# B&R Automation Studio project ABC_Pltzr (part 2)

#### bgTelnetSrvr-astcpV2.c
```c
#include <bur/plctypes.h>

#ifdef _DEFAULT_INCLUDES
	#include <AsDefault.h>
#endif
/*
File: bgTelnetSrvr-astcpV2.c
=====

Modified on June 2015:
-modifications and adjustements to the latest version of bglib and B&R libraries

Modified on Jyly 2007:
THIS IS AN UPDATED VERSION OF THE TELNET SERVER WITH A SUPPORT FOR NEW B&R TCP LIBRARY!
OLD B&R TCP LIBRARY: ETHERNET.LIB
NEW B&R TCP LIBRARY: ASTCP.LIB

B&R Libraries:
==============
Make sure to add following .a files to the task using this source file:
libsys_lib.a
libbrsystem.a
libastcp.a

About:
======
- this cyclic task is an implemenation of a telnet server for a B&R PCC
- when this task is active, it should be possible to connect remote telnet client to this PCC
- once the remote telnet client is connected, this task will start outputing debug messages
posted into the globaly defined RingBuffer structure
- following diagram shows the implemenation:

							+----------------->[ring buffer memory]
							|
					+-------*-------+
write to RingBuff	|gRingBuffer	|	read from RingBuff
			+------>|				|---------------+
			|		+---------------+				|
			|		global RingBuffer struct		|
			|										|
+=======+	|										|		+===============+
|task1	|-->+										+------>|bgtelnet		|---> if(telnet_client_is_connected)
+=======+	|												|(this task)	|		send_data_to_telnet_client
			|												+===============+
+=======+	|
|task2	|-->+
+=======+	|
			|
+=======+	|
|task3	|-->+
+=======+

- ring buffer memory is allocated at startup, and the size can be adjusted here (the default buffer size is 256kB)

WARNING: is the ring buffer memory is too small for the amount of data written into the buffer,
messages may get overwritten & lost!!!

- any task that needs to send debug messages via telnet needs following:

1) Include following at the top of the C module:
#include "bglib/bgdebug.h"

2) Within the code use following sprintf style debug function to define dbg messages
Examples:
a)
DBG("My debug message\n\r");

b)
{
int Value;
char Text[64];
strcpy(&Text[0], "Hello World\r\n");
DBG("Value=%d; Text=%s\n\r", Value, Text);
}

*/

/*
B&R components:
===============================================================================
*/
#include <bur/plc.h>
#include <bur/plctypes.h>
#include <astcp.h>
//#include <asstring.h>
#include <brsystem.h>
#include <sys_lib.h>

/*
BG components
===============================================================================
*/
#include "bgringbuffer.h"
#include "bgstring.h"
#include "../libraries/sprintf2/sprintf2.h"

/*Include required .c library files here. That way it's not needed in AS.*/
//#include "bgringbuffer.c"
//#include "bgsprintf.c"
//#include "bgstring.c"

#include "bgdebugV2.h"

/*Ring buffer size in bytes->adjust as needed*/
#define RB_SIZE 256000

/*User Private Library Error Numbers (value assigned as suggested in the B&R help file)*/
#define USER_ERROR_MIN  0xC350
#define USER_ERROR_MAX  0xEA5F
#define USER_ERROR_FTP  USER_ERROR_MIN + 10

/*telnet implemenation specifics*/
#define CMD_DONE	0
#define CMD_BUSY	1
#define CMD_ERROR	2

#define TELNET_SEND_BUFFER_SIZE 2048
#define TELNET_RECV_BUFFER_SIZE 256
#if 0
typedef struct bgSocketServer_typ{
	unsigned int sockStateData; 	/*state of the server data socket*/
	unsigned int telnetRecvState; 	/*state of the telnet server receiver*/
	unsigned int telnetSendState; 	/*state of the telnet server receiver*/

	unsigned int sockSendOk;

	int	cmdError;
	int	cmdErrorCode;

	char isConnected;
	char isLoggedIn;
	char isDataPortReady;

	char isEcho;

	char sockData_Timer;
	int sockData_TimerTime;
	int sockData_TimerCounter;

#if 0
/*following is used during development*/
	char devDataSendBuf[TELNET_SEND_BUFFER_SIZE];
	char devDataRecvBuf[TELNET_RECV_BUFFER_SIZE];
	char devLineRecvBuf[TELNET_RECV_BUFFER_SIZE];
#endif
	char *dataSendBuf;
	char *dataRecvBuf;
	char *lineRecvBuf;

	UDINT *ringDataBuffer;	/*ptr to allocated space used as a RingBuffer*/
	UDINT *sendRecvBuffer;	/*ptr to allocated space used for send/recv buffers*/

	char iacRecvBuf[10];

	DINT lineIndex;
	DINT lineIndexPrev;

	TcpOpen_typ TCPopen_1;
	TcpServer_typ TCPserv_1;
	TcpSend_typ TCPsend_1;
	TcpRecv_typ TCPrecv_1;
	TcpClose_typ TCPclose_1;
	TcpIoctl_typ TCPioctl_1;

	MEMInfo_typ MEMInfo;
	unsigned int memAllocStatus1;
	unsigned int memAllocStatus2;

	struct counter {
		int recv_frames;
		int iac;
		int lines;
		int send_frames;
	}counter;

	int test;
	int testCounter;
	STRING clientIpAddr[32];
	int delayCounter;
}bgSocketServer_typ;
#endif

/* Telnet protocol characters (don't change)*/
#define IAC     (255) /*"Interpret As Command"*/
#define DONT    (254)
#define DO      (253)
#define WONT    (252)
#define WILL    (251)
#define theNULL (0)

#define BS		(8)		/*0x8 - back space char*/
#define LF		(10)	/*0xa - line feed*/
#define CR		(13)	/*0xd - carrige return*/
#define EC      (247)  /*# Erase Character*/

/*telnet server related local PVs*/
//_LOCAL bgSocketServer_typ dbgTerm;

int bgSocketServerIsSendReady(bgSocketServer_typ *p);
int bgSocketServer(int init, bgSocketServer_typ *p);
void bgSocketServerRecv(bgSocketServer_typ *p);
void bgTelnetServerProcessCmd(bgSocketServer_typ *p, int length);
void bgTelnetServerProcessLine(bgSocketServer_typ *p);
void bgTelnetServerWelcomeMsg(bgSocketServer_typ *p);
void bgSocketServerSendData(bgSocketServer_typ *p, int len);
char* bgSocketGetSendBuffer(bgSocketServer_typ *p);
int bgSocketGetSendBufferSize(bgSocketServer_typ *p);
void bgTelnetSrvrMemAlloc(bgSocketServer_typ *p);
void bgTelnetServerCLI(bgSocketServer_typ *p);

void bgCLIHelp(bgSocketServer_typ *pTerm);

void bgCLIDebug(bgSocketServer_typ *pTerm, bgStringList_typ *p);
void bgCLIDebugHelp(bgSocketServer_typ *pTerm, bgStringList_typ *p);
void bgCLIDebugLevel(bgSocketServer_typ *pTerm, bgStringList_typ *p);
void bgCLIDebugFormat(bgSocketServer_typ *pTerm, bgStringList_typ *p);
void bgCLIDebugFilter(bgSocketServer_typ *pTerm, bgStringList_typ *p);

void bgCLIErrLog(bgSocketServer_typ *pTerm, bgStringList_typ *p);

void bgCLIPV(bgSocketServer_typ *pTerm, bgStringList_typ *p);
void bgCLIPVHelp(bgSocketServer_typ *pTerm, bgStringList_typ *p);
void bgCLIPVList(bgSocketServer_typ *pTerm, bgStringList_typ *p);
void bgCLIPVGet(bgSocketServer_typ *pTerm, bgStringList_typ *p);

const char *bgCLIGetPVTypeString(int pvTypeIndex);
void bgCLIPVPrintValue(bgSocketServer_typ *pTerm, unsigned int data_typ, unsigned int data_len, unsigned int dimension, unsigned int adr);

#if 0
_LOCAL char buffer[1024];
#endif

#define PV_TYPE_MAX_INDEX	15
static const char *bgPVTypeStrings[PV_TYPE_MAX_INDEX + 1]={
"STRUCT",
"BOOL  ",
"INT8  ",
"INT16 ",
"INT32 ",
"BYTE  ",
"WORD  ",
"LONG  ",
"FLOAT ",
"VISTR ",
"OCTET ",
"DATE  ",
"TIME  ",
"DIFF  ",
"BIT   ",
"ARRAY ",
};

static const char *bgDbgLevels[5]={
"CRITICAL",
"ERROR",
"WARNING",
"INFO",
"DEBUG",
};

/*
========================================================================================
*/
void bgTelnetSrvrInit(bgSocketServer_typ* pTerm, bgRingBuffer_typ* pRB)
{
	if(!pTerm || !pRB)
		return;

	/*allocate memory for ringBuffer and send/recv buffers*/
	bgTelnetSrvrMemAlloc(pTerm);

	/*init global RingBuffer*/
	bgRingBuffInit(pRB, (char*)pTerm->ringDataBuffer, RB_SIZE);
	pTerm->pRB = (UDINT)pRB;

	/*init telnet server*/
	bgSocketServer(1, pTerm);
}
/*
========================================================================================
*/
void bgTelnetSrvrCyclic(bgSocketServer_typ* pTerm)
{
int len;
bgRingBuffer_typ* pRB;

	if(!pTerm || !pTerm->pRB)
		return;

	pRB = (bgRingBuffer_typ*) (pTerm->pRB);

	/*if memalloc failed -> this task is useless*/
	if(pTerm->memAllocStatus1 || pTerm->memAllocStatus2)
		return;

	/*testing only; to enable it, use PV monitor to set variable > 10*/
	if(pTerm->testCounter > 10){
		pTerm->testCounter++;
		if(!(pTerm->testCounter % 10)){
			/*example of debug messages using different debug levels*/
			DBG(pRB, "DBG: Server Test Output %d\r\n", pTerm->testCounter);

			DBGCRT(pRB, "CRITICAL: Server Test Output %d\r\n", pTerm->testCounter);
			DBGERR(pRB, "ERROR: Server Test Output %d\r\n", pTerm->testCounter);
			DBGWAR(pRB, "WARNING: Server Test Output %d\r\n", pTerm->testCounter);
			DBGINF(pRB, "INFO: Server Test Output %d\r\n", pTerm->testCounter);
			DBGDBG(pRB, "DEBUG: Server Test Output %d\r\n", pTerm->testCounter);
		}
	}

	/*monitor if server is ready to send*/
	if( bgSocketServerIsSendReady(pTerm) ){
		/*get data from the ring buffer*/
		len = bgRingBuffGet( (bgRingBuffer_typ*) pTerm->pRB, bgSocketGetSendBuffer(pTerm), bgSocketGetSendBufferSize(pTerm) );

		if(len){
			/*send data*/
			bgSocketServerSendData(pTerm, len);
		}
	}

	/*execute server state machine cyclicly*/
    bgSocketServer(0, pTerm);
}

/*
========================================================================================
*/
void bgTelnetSrvrMemAlloc(bgSocketServer_typ *p)
{
unsigned int memSize;

	/*Get System Memory Information*/
	p->MEMInfo.enable = 1;
	MEMInfo(&p->MEMInfo);

/*TODO: use meminfo to see how much to allocated for ring buffer*/

	/*allocate space for RingBuffer data*/
	if(p->ringDataBuffer == 0){
		/* allocate new memory from RAM*/
    	p->memAllocStatus1 = TMP_alloc(RB_SIZE, (void**)&p->ringDataBuffer);
	}else{
		/*memory is allready allocated -> free it first!*/
    	p->memAllocStatus1 = TMP_free(RB_SIZE, (void**)p->ringDataBuffer);

    	/*allocate new memory from RAM*/
    	p->memAllocStatus1 = TMP_alloc(RB_SIZE, (void**)p->ringDataBuffer);
	}

	memSize = TELNET_SEND_BUFFER_SIZE + 2 * TELNET_RECV_BUFFER_SIZE;
	/*allocate space for send/recv buffers*/
	if(p->sendRecvBuffer == 0){
		/* allocate new memory from RAM*/
    	p->memAllocStatus2 = TMP_alloc(RB_SIZE, (void**)&p->sendRecvBuffer);
	}else{
		/*memory is allready allocated -> free it first!*/
    	p->memAllocStatus2 = TMP_free(RB_SIZE, (void**)p->sendRecvBuffer);

    	/*allocate new memory from RAM*/
    	p->memAllocStatus2 = TMP_alloc(RB_SIZE, (void**)p->sendRecvBuffer);
	}

	/*assign send/recv buffer ptrs*/
	p->dataSendBuf = (signed char*)p->sendRecvBuffer;
	p->dataRecvBuf = (signed char*)(p->sendRecvBuffer + TELNET_SEND_BUFFER_SIZE);
	p->lineRecvBuf = (signed char*)(p->sendRecvBuffer + TELNET_SEND_BUFFER_SIZE + TELNET_RECV_BUFFER_SIZE);

/*
Development only!
*/
/*
	p->dataSendBuf = (char*)p->devDataSendBuf;
	p->dataRecvBuf = (char*)p->devDataRecvBuf;
	p->lineRecvBuf = (char*)p->devLineRecvBuf;
*/
}

/*
========================================================================================
*/
#define TELNETD_STATE_NONE 0
#define TELNETD_STATE_INITOPEN 1
#define TELNETD_STATE_OPEN 2
#define TELNETD_STATE_SERVER 3
#define TELNETD_STATE_SEND 4
#define TELNETD_STATE_RECEIVE 5
#define TELNETD_STATE_CLOSE 6
#define TELNETD_STATE_CLOSE_DELAY 7

void bgSocketServerSendData(bgSocketServer_typ *p, int len)
{
	p->TCPsend_1.datalen = len;
	p->sockStateData = TELNETD_STATE_SEND;
}

char* bgSocketGetSendBuffer(bgSocketServer_typ *p)
{
	return ((char*)(p->dataSendBuf));
}

int bgSocketGetSendBufferSize(bgSocketServer_typ *p)
{
	return (TELNET_SEND_BUFFER_SIZE);
}

int bgSocketServerIsSendReady(bgSocketServer_typ *p)
{
	return(p->sockSendOk);
}

int bgSocketServer(int init, bgSocketServer_typ *p)
{
    /*open data socket (listen)*/
	if( (init == 1) && !p->sockStateData)
		p->sockStateData = 1;

    /*close data socket (listen stop)*/
	if( init == 2){
		/*command socket is telling us to receive data from server
		after this event, keep receiving until we don't get any data
		for a certain period of time
		*/
		p->sockData_Timer = 1;
		p->sockData_TimerTime = 10;
		p->sockData_TimerCounter = 0;
	}

	switch(p->sockStateData){
		case TELNETD_STATE_NONE:
    		return CMD_DONE;
		break;
		case TELNETD_STATE_INITOPEN:
			p->sockData_Timer = 0;
			p->isEcho = 1;
			p->lineIndex = 0;
			p->lineIndexPrev = 0;

			p->TCPopen_1.enable = 1;			/* port number of the server socket*/
			p->TCPopen_1.port = 23;				/* port number of the server socket*/
			p->TCPopen_1.pIfAddr = 0;
			p->TCPopen_1.options = tcpOPT_REUSEADDR;
    		p->sockStateData = TELNETD_STATE_OPEN;
		break;
		case TELNETD_STATE_OPEN:
			TcpOpen(&p->TCPopen_1);

			if( p->TCPopen_1.status == 0xFFFF )
				return CMD_BUSY;

			if( !p->TCPopen_1.status ){
				p->TCPserv_1.enable = 1;
				p->TCPserv_1.ident = p->TCPopen_1.ident;
				p->TCPserv_1.backlog = 0;
	    		p->TCPserv_1.pIpAddr = (UDINT)(p->clientIpAddr);
				p->sockStateData = TELNETD_STATE_SERVER;
				return CMD_BUSY;
			}

/* TODO: TcpOpen error handling! */
			p->sockStateData = TELNETD_STATE_NONE;
			p->isDataPortReady = 0;
		break;
		case TELNETD_STATE_SERVER:
    		TcpServer(&p->TCPserv_1);					/* makes a connection with the clients */

			if(p->TCPserv_1.status == 0xFFFF)
				return CMD_BUSY;

			if(!p->TCPserv_1.status){
				p->TCPsend_1.enable = 1;
   				p->TCPsend_1.ident = p->TCPserv_1.identclnt;   /* copy the  Ident number */
				p->TCPsend_1.flags = 0;
				p->TCPsend_1.pData = (UDINT)p->dataSendBuf;

   				p->TCPrecv_1.enable = 1;
   				p->TCPrecv_1.ident = p->TCPserv_1.identclnt;   /* copy the  Ident number */
   				p->TCPrecv_1.pData = (UDINT)p->dataRecvBuf; /* address of the buffer */;
   				p->TCPrecv_1.datamax = TELNET_RECV_BUFFER_SIZE; /* length of the buffer */;

	   			p->TCPclose_1.ident = p->TCPserv_1.identclnt;    /* copy the  Ident number */

    			p->sockStateData = TELNETD_STATE_RECEIVE;
				bgTelnetServerWelcomeMsg(p);
				return CMD_BUSY;
			}

/*TODO: what to do on error?*/
			goto errorExit;
		break;
		case TELNETD_STATE_SEND:
			p->sockSendOk = 0;
            TcpSend(&p->TCPsend_1);            				/* send the data */
            if(!p->TCPsend_1.status){
            	p->counter.send_frames++;
    			p->sockStateData = TELNETD_STATE_RECEIVE;
			}

			/*in case of the following error -> close connection*/
            if( (p->TCPsend_1.status == 27210) 	||
            	(p->TCPsend_1.status == 27135)	||
            	(p->TCPsend_1.status == tcpERR_NOT_CONNECTED)	||
            	(p->TCPsend_1.status == tcpERR_SYSTEM)	||
            	(p->TCPsend_1.status == 27249)
            ){
    			p->sockStateData = TELNETD_STATE_CLOSE;
			}
		break;
		case TELNETD_STATE_RECEIVE:
            TcpRecv(&p->TCPrecv_1);          				/* recv data*/

            if(!p->TCPrecv_1.status){
            	p->counter.recv_frames++;
                if(p->TCPrecv_1.recvlen){
                    bgSocketServerRecv(p);
                }else{
					/*remote socket has closed*/
    				p->sockStateData = TELNETD_STATE_CLOSE;    /*close this server socket*/
				}
            }else{
    			p->sockSendOk = 1;							/*enable others to send*/
            }

		break;
		case TELNETD_STATE_CLOSE:
			p->TCPclose_1.enable = 1;
			p->TCPclose_1.how = tcpSHUT_RD & tcpSHUT_WR;

            TcpClose(&p->TCPclose_1);          				/* set the socket free */

			if(p->TCPclose_1.status == 0xFFFF){
				return CMD_BUSY;
			}

			p->delayCounter = 10;
	    	p->sockStateData = TELNETD_STATE_CLOSE_DELAY;
		break;
		case TELNETD_STATE_CLOSE_DELAY:
			p->delayCounter--;
			if(!p->delayCounter){
	    		p->sockStateData = TELNETD_STATE_SERVER;
				p->isDataPortReady = 0;
				p->sockData_Timer = 0;
			}

		break;
		default:
		break;
		}

    return CMD_BUSY;

errorExit:

    TcpClose(&p->TCPclose_1);          /* set the socket free */
	p->sockStateData = 1;
	p->isDataPortReady = 0;
	return CMD_ERROR;
}

void bgSocketServerRecv(bgSocketServer_typ *p){

int len = p->TCPrecv_1.recvlen;
int i, k;
unsigned char dataChr;

bgRingBuffer_typ* pRB = (bgRingBuffer_typ*) (p->pRB);
//DBG(pRB, "DBG: Server Test Output %d\r\n", pTerm->testCounter);

	for(i=0, k=0;i<len;i++){
		dataChr = p->dataRecvBuf[i];

		switch(p->telnetRecvState){
			case 0:/*normal receive; check for telnet command chars*/

				/*0 - NOP*/
				if( dataChr == theNULL )
					break;

				/*"Interpret As Command"?*/
				if( dataChr == IAC ){
					p->iacRecvBuf[0] = dataChr;
					p->telnetRecvState++;
				}else
				if( (dataChr == BS) && p->lineIndex ){
					p->lineIndex--;
					p->lineIndexPrev = p->lineIndex;
					DBGMSG(pRB, "%c", BS);
				}else
				if( (dataChr == BS) && !p->lineIndex ){
					p->lineIndexPrev = p->lineIndex;
				}else{

					/*regular char -> store into the line rcv buffer*/
					p->lineRecvBuf[p->lineIndex++] = dataChr;

					/*LineFeed or Carrige Return? -> EOL (End of Line)*/
					if( dataChr == LF )
						bgTelnetServerProcessLine(p);

					/*limit input -> overflow is danger!!!*/
					if( p->lineIndex >= (TELNET_RECV_BUFFER_SIZE - 5) )
						bgTelnetServerProcessLine(p);
				}
			break;
			case 1:/*get 2.nd telnet command char; <type of operation>*/

				/*check if there is a third char in command or not!?*/
				if( (dataChr >= WILL) && (dataChr <= DONT) ){
					p->iacRecvBuf[1] = dataChr;
					p->telnetRecvState++;
				}else{
					p->iacRecvBuf[1] = dataChr;
					p->telnetRecvState = 0;
					bgTelnetServerProcessCmd(p, 2);
				}

			break;
			case 2:/*get 3.rd telnet command char; <option>*/

				p->iacRecvBuf[2] = dataChr;
				p->telnetRecvState = 0;
				bgTelnetServerProcessCmd(p, 3);

			break;

		}
	}

	if(p->isEcho && (p->lineIndex > p->lineIndexPrev) ){
		int chrCount = p->lineIndex - p->lineIndexPrev;
		brsmemcpy((UDINT)p->dataSendBuf, (UDINT)(&p->lineRecvBuf[p->lineIndexPrev]), (UDINT)chrCount);
		bgSocketServerSendData(p, chrCount);
		p->lineIndexPrev = p->lineIndex;
	}

}

void bgTelnetServerProcessCmd(bgSocketServer_typ *p, int length)
{
	p->counter.iac++;
}

void bgTelnetServerProcessLine(bgSocketServer_typ *p)
{
bgRingBuffer_typ* pRB = (bgRingBuffer_typ*) (p->pRB);

	p->counter.lines++;

	bgTelnetServerCLI(p);

	p->lineIndex = 0;
	p->lineIndexPrev = 0;

	DBGMSG(pRB, "\r\n>");
}

void bgTelnetServerWelcomeMsg(bgSocketServer_typ *p)
{
bgRingBuffer_typ* pRB = (bgRingBuffer_typ*) (p->pRB);

	DBGMSG(pRB, "###########################################################\r\n");
	DBGMSG(pRB, "#                 Welcome!                                #\r\n");
	DBGMSG(pRB, "#Debug and Command Interface to B&R controller via Telnet.#\r\n");
	DBGMSG(pRB, "#Type '?' or 'help' for more information.                 #\r\n");
	DBGMSG(pRB, "###########################################################\r\n");
	DBGMSG(pRB, "#Connection from: %s", p->clientIpAddr);
	DBGMSG(pRB, "###########################################################\r\n");
	DBGMSG(pRB, "\r\n>");
}

void bgTelnetServerCLI(bgSocketServer_typ *p)
{
int lineLen = p->lineIndex - 1;
char *pLine;
char *pWord;
bgStringList_typ listOfWordsInLine;
int wordCount;
bgRingBuffer_typ* pRB = (bgRingBuffer_typ*) (p->pRB);

	/*terminate received line with 0 -> line is now a "C" string */
	p->lineRecvBuf[lineLen] = 0;

#if 0
	/*for AS watch window*/
	strcpy(buffer, p->lineRecvBuf);
#endif

	/*check if CR present in line*/
	if(lineLen && (p->lineRecvBuf[lineLen-1] == CR) ){
		lineLen--;
		p->lineRecvBuf[lineLen] = 0;
	}

	if( !lineLen )
		return;

#if 0
	DBG(pRB, "\n\rCLI: Len=[%d],  Line=[%s]\n\r", lineLen, p->lineRecvBuf);
#endif

	/*line is received!*/
	pLine = (char*)(p->lineRecvBuf);

	/*split line into list of words*/
	listOfWordsInLine.src = (unsigned char*)pLine;
	wordCount = bgStringSplitLine(&listOfWordsInLine, ' ');

	if( wordCount == 0)
		return;

/*
#############################################################################################
#############################################################################################
*/

	/*first word -> command*/
	pWord = bgStringLower((char*)listOfWordsInLine.items[0]);

	/*if first character is '#'->comment, nothing to do*/
	if( *pWord == '#' ){
		return;
	}

	/*search for commands*/
	if( bgStringIsMatch(pWord, "?", 1) ){
		bgCLIHelp(p);
		return;
	}

	if( bgStringIsMatch(pWord, "help", 1) ){
		bgCLIHelp(p);
		return;
	}

	if( bgStringIsMatch(pWord, "debug", 1) ){
		bgCLIDebug(p, &listOfWordsInLine);
		return;
	}

	if( bgStringIsMatch(pWord, "errlog", 1) ){
		bgCLIErrLog(p, &listOfWordsInLine);
		return;
	}

	if( bgStringIsMatch(pWord, "pv", 1) ){
		bgCLIPV(p, &listOfWordsInLine);
		return;
	}

	DBGMSG(pRB, "\n\rUnknown command!\n\rPlease type '?' for list of valid commands!\r\n");

}

/*
#############################################################################################
#############################################################################################
help
#############################################################################################
#############################################################################################
*/
void bgCLIHelp(bgSocketServer_typ *pTerm)
{
bgRingBuffer_typ* pRB = (bgRingBuffer_typ*) (pTerm->pRB);

	DBGMSG(pRB, "\r\n");
	DBGMSG(pRB, "###########################################################\r\n");
	DBGMSG(pRB, "#Debug and Command Interface to B&R controller via Telnet.#\r\n");
	DBGMSG(pRB, "#Version: 1.0                                             #\r\n");
	DBGMSG(pRB, "#Date   : 2005-10-01                                      #\r\n");
	DBGMSG(pRB, "#Author : Belgor Inc.                                     #\r\n\r\n");
	DBGMSG(pRB, "#Available commands:                                      #\r\n");
	DBGMSG(pRB, "# ?, help  - display this help text                       #\r\n");
	DBGMSG(pRB, "# debug    - adjust & control debug output                #\r\n");
	DBGMSG(pRB, "# errlog   - display controller's error log entries       #\r\n");
	DBGMSG(pRB, "# pv       - access application's PVs (Process Variables) #\r\n");
	DBGMSG(pRB, "# '#'      - comment (line starting with '#' is ignored)  #\r\n\r\n");
	DBGMSG(pRB, "#For more information about individual commands type:     #\r\n");
	DBGMSG(pRB, "#<CommandName> ?                                          #\r\n");
	DBGMSG(pRB, "#or                                                       #\r\n");
	DBGMSG(pRB, "#<CommandName> help                                       #\r\n");
	DBGMSG(pRB, "###########################################################\r\n");
	DBGMSG(pRB, "\r\n");
}

/*
#############################################################################################
#############################################################################################
debug
#############################################################################################
#############################################################################################
*/
void bgCLIDebug(bgSocketServer_typ *pTerm, bgStringList_typ *p)
{

int cliParamIndex;
char *pWord;
//bgRingBuffer_typ* pRB = (bgRingBuffer_typ*) (pTerm->pRB);

	cliParamIndex = 1;

	if( p->itemCount <= cliParamIndex ){
		bgCLIDebugHelp(pTerm, p);
		return;
	}

	pWord = bgStringLower( (char*)( p->items[cliParamIndex]) );

	if( bgStringIsMatch(pWord, "?", 1) ){
		bgCLIDebugHelp(pTerm, p);
		return;
	}

	if( bgStringIsMatch(pWord, "help", 1) ){
		bgCLIDebugHelp(pTerm, p);
		return;
	}

	if( bgStringIsMatch(pWord, "level", 1) ){
		bgCLIDebugLevel(pTerm, p);
		return;
	}

	if( bgStringIsMatch(pWord, "format", 1) ){
		bgCLIDebugFormat(pTerm, p);
		return;
	}

	if( bgStringIsMatch(pWord, "filter", 1) ){
		bgCLIDebugFilter(pTerm, p);
		return;
	}

	bgCLIDebugHelp(pTerm, p);

}

/*
>debug ?
>debug help
*/
void bgCLIDebugHelp(bgSocketServer_typ *pTerm, bgStringList_typ *p)
{
bgRingBuffer_typ* pRB = (bgRingBuffer_typ*) (pTerm->pRB);

	DBGMSG(pRB, "\r\n");
	DBGMSG(pRB, "Command: debug\n\r");
	DBGMSG(pRB, "===========================================================\n\r");
	DBGMSG(pRB, "- adjust and control debug output\r\n");
	DBGMSG(pRB, "Following is the list of valid 'debug' commands:\r\n\r\n");
	DBGMSG(pRB, " debug\r\n");
	DBGMSG(pRB, " debug ?\r\n");
	DBGMSG(pRB, " debug help\r\n");
	DBGMSG(pRB, " --- displays this message\r\n\r\n");
	DBGMSG(pRB, " debug level\r\n");
	DBGMSG(pRB, " --- display current debug level, change (set) debug level\r\n\r\n");
	DBGMSG(pRB, " debug format\r\n");
	DBGMSG(pRB, " --- display current debug format, change (set) debug format\r\n");
	DBGMSG(pRB, "===========================================================\n\r");
	DBGMSG(pRB, "\r\n");
}

/*
>debug level
*/
void bgCLIDebugLevel(bgSocketServer_typ *pTerm, bgStringList_typ *p)
{
unsigned int value;
bgRingBuffer_typ* pRB = (bgRingBuffer_typ*) (pTerm->pRB);

	if( p->itemCount <= 2){
		if( pRB->dbgLevel > BG_DEBUG_LEVEL_DEBUG )
			pRB->dbgLevel = 0;

		DBGMSG(pRB, "\n\rCurrent Debug Level : %d (%s)\r\n", pRB->dbgLevel, bgDbgLevels[pRB->dbgLevel]);
		goto Exit;
	}

	if( bgAsciiToUint( (char*)(p->items[2]), &value) ){

		if( value <= BG_DEBUG_LEVEL_DEBUG){
			DBGMSG(pRB, "\n\rCurrent Debug Level : %d (%s)\r\n", pRB->dbgLevel, bgDbgLevels[pRB->dbgLevel]);
			pRB->dbgLevel = value;
			    DBGMSG(pRB, "New Debug Level     : %d (%s)\r\n", pRB->dbgLevel, bgDbgLevels[pRB->dbgLevel]);
			return;
		}else{
			DBGMSG(pRB, "\n\rCurrent Debug Level : %d (%s)\r\n", pRB->dbgLevel, bgDbgLevels[pRB->dbgLevel]);
			DBGMSG(pRB, "\n\rInput Parameter Error! Debug Level value '%d' out of range!\r\n", value);
			goto Exit;
		}

	}else{

		DBGMSG(pRB, "\n\rInput Parameter Error! Entered value '%s' not a numeric string!\r\n", p->items[2]);
		goto Exit;

	}

Exit:

		DBGMSG(pRB, "\n\rPossible Debug Levels are:\r\n");
		DBGMSG(pRB, "0 - CRITICAL\n\r");
		DBGMSG(pRB, "1 - ERROR\n\r");
 		DBGMSG(pRB, "2 - WARNING\n\r");
		DBGMSG(pRB, "3 - INFO\n\r");
		DBGMSG(pRB, "4 - DEBUG\n\r");
		DBGMSG(pRB, "\n\r");
		DBGMSG(pRB, "To set debug level use:\n\r");
		DBGMSG(pRB, "debug level [0|1|2|3|4]\n\r");
		DBGMSG(pRB, "\n\r");
		DBGMSG(pRB, "Example (Setting debug level to 4 = DEBUG):\n\r");
		DBGMSG(pRB, "debug level 4\n\r");

}

/*
>debug format
*/
void bgCLIDebugFormat(bgSocketServer_typ *pTerm, bgStringList_typ *p)
{
unsigned int value;
bgRingBuffer_typ* pRB = (bgRingBuffer_typ*) (pTerm->pRB);

	if( p->itemCount <= 2){
		DBGMSG(pRB, "\n\rCurrent Debug Format : %x\r\n", pRB->dbgFormat);
		goto Exit;
	}

	if( bgAsciiToUint( (char*)p->items[2], &value) ){
		DBGMSG(pRB, "\n\rCurrent Debug Format : %x\r\n", pRB->dbgFormat);
		pRB->dbgFormat = value;
		    DBGMSG(pRB, "New Debug Format     : %x\r\n", pRB->dbgFormat);
		return;
	}else{

		DBGMSG(pRB, "\n\rInput Parameter Error! Entered value '%s' not a numeric string!\r\n", p->items[2]);
		goto Exit;

	}

Exit:

		DBGMSG(pRB, "\n\rDebug Format Value is a bit field with following fields:\r\n");
		DBGMSG(pRB, "Bit[0] - FileName     (0-off, 1-on)\n\r");
		DBGMSG(pRB, "Bit[1] - FunctionName (0-off, 1-on)\n\r");
		DBGMSG(pRB, "Bit[2] - TimeStamp    (0-off, 1-on)\n\r");
		DBGMSG(pRB, "Bit[3] - Level        (0-off, 1-on)\n\r");
		DBGMSG(pRB, "\n\r");
		DBGMSG(pRB, "To set debug format value use:\n\r");
		DBGMSG(pRB, "debug format [value]");
		DBGMSG(pRB, "\n\r");
		DBGMSG(pRB, "Example (Set debug format to 3 (bit[0]=1, bit[1]=1) -> Enable FileName and FunctionName display:\n\r");
		DBGMSG(pRB, "debug format 3\n\r");
}

/*
>debug filter
*/
void bgCLIDebugFilter(bgSocketServer_typ *pTerm, bgStringList_typ *p)
{
bgRingBuffer_typ* pRB = (bgRingBuffer_typ*) (pTerm->pRB);
	DBGMSG(pRB, "\n\rCmd='debug filter' TODO!\r\n");
}
/*
#############################################################################################
#############################################################################################
errlog
#############################################################################################
#############################################################################################
*/
void bgCLIErrLog(bgSocketServer_typ *pTerm, bgStringList_typ *p)
{
ERR_xtyp errStruct;
int i;
unsigned int status;
bgRingBuffer_typ* pRB = (bgRingBuffer_typ*) (pTerm->pRB);

	DBGMSG(pRB, "\n\rList Error Log Entries\n\r\n\r");
	DBGMSG(pRB, "=============================================================+==========\n\r\n\r");
	DBGMSG(pRB, "#  | Time stamp             | Errno | ErrInfo    | T | Task  | \n\r");
	DBGMSG(pRB, "---+------------------------+-------+------------+---+-------+----------\n\r");
/*	DBGMSG("01 | 2005/09/21 12:50:30.44 | 12345 | 0x12345678 | 1 | syslog| \n\r");*/
/*  DBGMSG("[%02d] | %s | %05d | 0x%08x | %d | '%s' | '%s'\n\r"*/

	for(i=0;i<10;i++){
		status = ERRxread(i, &errStruct);
		if(!status){
			char timeStamp[64];
			/*bgsprintf*/sprintf2(timeStamp, "%04d/%02d/%02d %02d:%02d:%02d.%02d",
				errStruct.err_year,
				errStruct.err_month,
				errStruct.err_day,
				errStruct.err_hour,
				errStruct.err_minute,
				errStruct.err_second,
				errStruct.err_millisec);

			DBGMSG(pRB, "%02d | %s | %05d | 0x%08x | %d | '%s' | '%s'\n\r",
			i, timeStamp, errStruct.err_nr, errStruct.err_info, errStruct.err_type, errStruct.t_name, errStruct.err_string);
		}
	}
}

/*
#############################################################################################
#############################################################################################
pv
#############################################################################################
#############################################################################################
*/
void bgCLIPV(bgSocketServer_typ *pTerm, bgStringList_typ *p)
{
int cliParamIndex;
//bgRingBuffer_typ* pRB = (bgRingBuffer_typ*) (pTerm->pRB);

	cliParamIndex = 1;

	if( p->itemCount <= cliParamIndex ){
		bgCLIPVHelp(pTerm, p);
		return;
	}

	if( bgStringIsMatch( (char*)(p->items[cliParamIndex]), "?", 1) ){
		bgCLIPVHelp(pTerm, p);
		return;
	}

	if( bgStringIsMatch((char*)(p->items[cliParamIndex]), "help", 1) ){
		bgCLIPVHelp(pTerm, p);
		return;
	}

	if( bgStringIsMatch((char*)(p->items[cliParamIndex]), "list", 1) ){
		bgCLIPVList(pTerm, p);
		return;
	}

	if( bgStringIsMatch((char*)(p->items[cliParamIndex]), "get", 1) ){
		bgCLIPVGet(pTerm, p);
		return;
	}

	bgCLIPVHelp(pTerm, p);
}

/*
>pv ?
>pv help
*/
void bgCLIPVHelp(bgSocketServer_typ *pTerm, bgStringList_typ *p)
{
bgRingBuffer_typ* pRB = (bgRingBuffer_typ*) (pTerm->pRB);

	DBGMSG(pRB, "\r\n");
	DBGMSG(pRB, "Command: pv\n\r");
	DBGMSG(pRB, "===========================================================\n\r");
	DBGMSG(pRB, "- list, get and set application PVs (Process Variables)\r\n");
	DBGMSG(pRB, "Following is the list of valid 'pv' commands:\r\n\r\n");
	DBGMSG(pRB, " pv ?\r\n");
	DBGMSG(pRB, " pv help\r\n");
	DBGMSG(pRB, " --- display this message\r\n");
	DBGMSG(pRB, " pv list\r\n");
	DBGMSG(pRB, " --- display list of available PVs in the system\r\n");
	DBGMSG(pRB, " pv get\r\n");
	DBGMSG(pRB, " --- get current value of a PV\r\n");
	DBGMSG(pRB, " pv set\r\n");
	DBGMSG(pRB, " --- set value of a PV\r\n");
	DBGMSG(pRB, "===========================================================\n\r");
	DBGMSG(pRB, "\r\n");
}

/*
>pv list
*/
void bgCLIPVList(bgSocketServer_typ *pTerm, bgStringList_typ *p)
{
PV_xList_typ pvxList;
int i;
unsigned int status;
unsigned int prev_index;
unsigned int next_index;
bgRingBuffer_typ* pRB = (bgRingBuffer_typ*) (pTerm->pRB);

	DBGMSG(pRB, "\n\rPV List:\n\r\n\r");
	DBGMSG(pRB, "==========================================================\n\r");
	DBGMSG(pRB, "#    | Type   | Len  | Dim  | Address    | Name\n\r");
	DBGMSG(pRB, "-----+--------+------+------+------------+----------------\n\r");
	prev_index = 0xFFFF;
	for(i=0; i<50; i++){
//UINT PV_xlist		(UINT prev_index, UINT *index, PV_xList_typ *pvl_p);
		status = PV_xlist((UINT)prev_index, (UINT*)&next_index, &pvxList);
		prev_index = next_index;

		if(!status){
			DBGMSG(pRB, "%4d | %s | %4d | %4d | 0x%08x | %s\n\r",
				i,  bgCLIGetPVTypeString(pvxList.data_typ), pvxList.data_len, pvxList.dimension, pvxList.adress,  pvxList.name);
		}else
			return;
	}
}

/*
>pv get
*/
void bgCLIPVGet(bgSocketServer_typ *pTerm, bgStringList_typ *p)
{
int cliParamIndex;
unsigned int status;
UDINT data_typ;
UDINT data_len;
UINT dimension;
UDINT adr;
bgRingBuffer_typ* pRB = (bgRingBuffer_typ*) (pTerm->pRB);

	cliParamIndex = 2;

	if( p->itemCount <= cliParamIndex )
		return;

//UINT PV_ninfo		(char *pv_name, UDINT *data_typ_p, UDINT *data_len_p, UINT *dimension_p);
	status = PV_ninfo((char*)(p->items[cliParamIndex]), (UDINT*)(&data_typ), (UDINT*)(&data_len), (UINT*)(&dimension));

	if( status ){
		DBGMSG(pRB, "\n\rError! Can't GET value for PV='%s'; Error#=%d\n\r", p->items[cliParamIndex], status);
		return;
	}

//UINT PV_xgetadr		(char *pv_name, UDINT *pv_adresse, UDINT *data_len);
	status = PV_xgetadr((char*)(p->items[cliParamIndex]), (UDINT*)(&adr), (UDINT*)(&data_len));

	if( status ){
		DBG(pRB, "Can't GET address for PV='%s'; Error=%d\n\r", p->items[cliParamIndex], status);
		return;
	}

	DBGMSG(pRB, "\n\r=========================================================\n\r");
	DBGMSG(pRB, "\n\rGet PV Value\n\r");
	DBGMSG(pRB, "=========================================================\n\r");
	DBGMSG(pRB, "PV='%s' Type=%s Len=%d Dim=%d Address=0x%08x\n\r",
			p->items[cliParamIndex], bgCLIGetPVTypeString(data_typ), data_len, dimension, adr);

	bgCLIPVPrintValue(pTerm, data_typ, data_len, dimension, adr);

}

void bgCLIPVPrintValue(bgSocketServer_typ* pTerm, unsigned int data_typ, unsigned int data_len, unsigned int dimension, unsigned int adr)
{
bgRingBuffer_typ* pRB = (bgRingBuffer_typ*) (pTerm->pRB);
/*
	if( dimension != 1)
		DBGMSG("TODO: display multidimensional values...");
*/
	switch(data_typ){
		case PB_DT_STRUCT:
			DBGMSG(pRB, "TODO: display struct values...");
		break;
		case PB_DT_BOOL:
			DBGMSG(pRB, "Value=%d", *( (char*)adr ));
		break;
		case PB_DT_INT8:
			DBGMSG(pRB, "Value=%d, (0x%x)", *( (char*)adr), *( (char*)adr ) );
		break;
		case PB_DT_INT16:
			DBGMSG(pRB, "Value=%d, (0x%x)", *( (short*)adr ), *( (short*)adr ) );
		break;
		case PB_DT_INT32:
			DBGMSG(pRB, "Value=%d, (0x%x)", *( (int*)adr ), *( (int*)adr ));
		break;
		case PB_DT_BYTE:
			DBGMSG(pRB, "Value=%u, (0x%x)", *( (unsigned char*)adr), *( (unsigned char*)adr ));
		break;
		case PB_DT_WORD:
			DBGMSG(pRB, "Value=%u, (0x%x)", *( (unsigned short*)adr), *( (unsigned short*)adr ));
		break;
		case PB_DT_LONG:
			DBGMSG(pRB, "Value=%u, (0x%x)", *( (unsigned int*)adr), *( (unsigned int*)adr ));
		break;
		case PB_DT_FLOAT:
			DBGMSG(pRB, "TODO: display float values...");
		break;
		case PB_DT_VIS:
			DBGMSG(pRB, "Value='%s'", (char*)adr );
		break;
		case PB_DT_OCTET:
			DBGMSG(pRB, "TODO: display octet values...");
		break;
		case PB_DT_DATE:
			DBGMSG(pRB, "TODO: display date values...");
		break;
		case PB_DT_TIME:
			DBGMSG(pRB, "TODO: display time values...");
		break;
		case PB_DT_DIFF:
			DBGMSG(pRB, "TODO: display time-diff values...");
		break;
		case PB_DT_BIT:
			DBGMSG(pRB, "TODO: display bit values...");
		break;
		case PB_DT_ARRAY:
			DBGMSG(pRB, "TODO: display array values...");
		break;
	}
}

#if 0
  status_adr = PV_xgetadr("PV_var1", &pv_adr, &data_len);   /* get the address
                                                             and the lenght of  PV */
  strcpy(PV_var2.name, "This is a test");       /* copy the string into PV */
  memcpy((UDINT*)pv_adr, &PV_var2, sizeof(PV_test));  /* copy the second to the first PV */
  status_item = PV_item("PV_var1", 0, itemname);      /* info of the first item of PV1 */
  status_ninfo = PV_ninfo("PV_var2", &data_typ, &data_len2, &dimension);/* info of PV2 */

#endif

const char *bgCLIGetPVTypeString(int pvTypeIndex){
	if(pvTypeIndex >= PV_TYPE_MAX_INDEX){
		return "TYPE=?";
	}

	return bgPVTypeStrings[pvTypeIndex];
}

/*
TELNET CONSTANTS
#######################################################################################################################
*/
#if 0
#define SE      (240)  /*# Subnegotiation End*/
#define NOP     (241)  /*# No Operation*/
#define DM      (242)  /*# Data Mark*/
#define BRK     (243)  /*# Break*/
#define IP      (244)  /*# Interrupt process*/
#define AO      (245)  /*# Abort output*/
#define AYT     (246)  /*# Are You There*/
#define EC      (247)  /*# Erase Character*/
#define EL      (248)  /*# Erase Line*/
#define GA      (249)  /*# Go Ahead*/
#define SB      (250)  /*# Subnegotiation Begin*/

/*
# Telnet protocol options code (don't change)
# These ones all come from arpa/telnet.h
*/
#define BINARY  (0) /*# 8-bit data path*/
#define ECHO    (1) /*# echo*/
#define RCP     (2) /*# prepare to reconnect*/
#define SGA     (3) /*# suppress go ahead*/
#define NAMS    (4) /*# approximate message size*/
#define STATUS  (5) /*# give status*/
#define TM      (6) /*# timing mark*/
#define RCTE    (7) /*# remote controlled transmission and echo*/
#define NAOL    (8) /*# negotiate about output line width*/
#define NAOP    (9) /*# negotiate about output page size*/
#define NAOCRD  (10) /*# negotiate about CR disposition*/
#define NAOHTS  (11) /*# negotiate about horizontal tabstops*/
#define NAOHTD  (12) /*# negotiate about horizontal tab disposition*/
#define NAOFFD  (13) /*# negotiate about formfeed disposition*/
#define NAOVTS  (14) /*# negotiate about vertical tab stops*/
#define NAOVTD  (15) /*# negotiate about vertical tab disposition*/
#define NAOLFD  (16) /*# negotiate about output LF disposition*/
#define XASCII  (17) /*# extended ascii character set*/
#define LOGOUT  (18) /*# force logout*/
#define BM      (19) /*# byte macro*/
#define DET     (20) /*# data entry terminal*/
#define SUPDUP  (21) /*# supdup protocol*/
#define SUPDUPOUTPUT  (22) /*# supdup output*/
#define SNDLOC  (23) /*# send location*/
#define TTYPE   (24) /*# terminal type*/
#define EOR     (25) /*# end or record*/
#define TUID    (26) /*# TACACS user identification*/
#define OUTMRK  (27) /*# output marking*/
#define TTYLOC  (28) /*# terminal location number*/
#define VT3270REGIME  (29) /*# 3270 regime*/
#define X3PAD   (30) /*# X.3 PAD*/
#define NAWS    (31) /*# window size*/
#define TSPEED  (32) /*# terminal speed*/
#define LFLOW   (33) /*# remote flow control*/
#define LINEMODE    (34) /*# Linemode option*/
#define XDISPLOC    (35) /*# X Display Location*/
#define OLD_ENVIRON (36) /*# Old - Environment variables*/
#define AUTHENTICATION  (37) /*# Authenticate*/
#define ENCRYPT (38) /*# Encryption option*/
#define NEW_ENVIRON (39) /*# New - Environment variables*/
/*
# the following ones come from
# http://www.iana.org/assignments/telnet-options
# Unfortunately, that document does not assign identifiers
# to all of them, so we are making them up
*/
#define TN3270E     (40) /*# TN3270E*/
#define XAUTH       (41) /*# XAUTH*/
#define CHARSET     (42) /*# CHARSET*/
#define RSP         (43) /*# Telnet Remote Serial Port*/
#define COM_PORT_OPTION     (44) /*# Com Port Control Option*/
#define SUPPRESS_LOCAL_ECHO (45) /*# Telnet Suppress Local Echo*/
#define TLS         (46) /*# Telnet Start TLS*/
#define KERMIT      (47) /*# KERMIT*/
#define SEND_URL    (48) /*# SEND-URL*/
#define FORWARD_X   (49) /*# FORWARD_X*/
#define PRAGMA_LOGON    (138) /*# TELOPT PRAGMA LOGON*/
#define SSPI_LOGON      (139) /*# TELOPT SSPI LOGON*/
#define PRAGMA_HEARTBEAT  (140) /*# TELOPT PRAGMA HEARTBEAT*/
#define EXOPL       (255) /*# Extended-Options-List*/
#define NOOPT       (0)     /**/
#endif
/*
TELNET INFO
#######################################################################################################################

The Network Virtual Terminal:
============================
Communication is established using TCP/IP and is based on a Network Virtual Terminal (NVT). On the
client, the Telnet program is responsible for translating incoming NVT codes to codes understood
by the client's display device as well as for translating client-generated keyboard codes into outgoing
NVT codes.

The NVT uses 7-bit codes for characters. The display device, referred to as a printer in the RFC, is
only required to display the standard printing ASCII characters represented by 7-bit codes and to
recognize and process certain control codes. The 7-bit characters are transmitted as 8-bit bytes with
the most significant bit set to zero. An end-of-line is transmitted as a carriage return (CR) followed
by a line feed (LF). If you want to transmit an actual carriage return, this is transmitted as a
carriage return followed by a NUL (all bits zero) character.

NVT ASCII is used by many other Internet protocols like SMTP and FTP.

The following control codes are required to be understood by the NVT.

Name            Code    Decimal Value   Function
=================================================
NULL            NUL     0               No operation
Line Feed       LF      10              Moves the printer to the next print line, keeping the same horizontal position.
Carriage Return CR      13              Moves the printer to the left margin of the current line.

The following further control codes are optional but should have the indicated defined effect on the
display.

Name            Code    Decimal Value Function
==============================================
BELL            BEL     7       Produces an audible or visible signal (which does NOT move the print head.
Back Space      BS      8       Moves the print head one character position towards the left margin. (On a printing device, this mechanism was commonly used to form composite characters by printing two basic characters on top of each other.)
Horizontal Tab  HT      9       Moves the printer to the next horizontal tab stop. It remains unspecified how either party determines or establishes where such tab stops are located.
Vertical Tab    VT      11      Moves the printer to the next vertical tab stop. It remains unspecified how either party determines or establishes where such tab stops are located.
Form Feed       FF      12      Moves the printer to the top of the next page, keeping the same horizontal position. (On visual displays, this commonly clears the screen and moves the cursor to the top left corner.)

The NVT keyboard is specified as being capable of generating all 128 ASCII codes by using keys, key
combinations, or key sequences

Commands:
=========
The Telnet protocol uses various commands to control the client-server connection. These commands are
transmitted within the data stream. The commands are distinguished from the data by setting the most
significant bit to 1. (Remember that data is transmitted as 7-bits with the eighth bit set to 0)
Commands are always introduced by the Interpret as command (IAC) character.

Here is the complete set of commands:

Name        Decimal Code    Meaning Comment
===========================================
SE          240             End of subnegotiation parameters
NOP         241             No operation
DM          242             Data mark Indicates the position of a Synch event within the data stream. This should always be accompanied by a TCP urgent notification.
BRK         243             Break Indicates that the "break" or "attention" key was hi.
IP          244             Suspend Interrupt or abort the process to which the NVT is connected.
AO          245             Abort output Allows the current process to run to completion but does not send its output to the user.
AYT         246             Are you there Send back to the NVT some visible evidence that the AYT was received.
EC          247             Erase character The receiver should delete the last preceding undeleted character from the data stream.
EL          248             Erase line Delete characters from the data stream back to but not including the previous CRLF.
GA          249             Go ahead Under certain circumstances used to tell the other end that it can transmit.
SB          250             Subnegotiation Subnegotiation of the indicated option follows.
WILL        251             will Indicates the desire to begin performing, or confirmation that you are now performing, the indicated option.
WONT        252             wont Indicates the refusal to perform, or continue performing, the indicated option.
DO          253             do Indicates the request that the other party perform, or confirmation that you are expecting the other party to perform, the indicated option.
DONT        254             dont Indicates the demand that the other party stop performing, or confirmation that you are no longer expecting the other party to perform, the indicated option.
IAC         255             Interpret as command Interpret as a command

Telnet Options:
===============
Options give the client and server a common view of the connection. They can be negotiated at any time during the
connection by the use of commands. They are described in separate RFCs.

The following are examples of common options:

Either end of a telnet dialogue can enable or disable an option either locally or remotely.
The initiator sends a 3 byte command of the form

    IAC,<type of operation>,<option>

The response is of the same form.

Operation is one of

Description     Decimal Code    Action
======================================
WILL            251             Sender wants to do something.
DO              252             Sender wants the other end to do something.
WONT            253             Sender doesn't want to do something.
DONT            254             Sender wants the other not to do something.

Associated with each of the these there are various possible responses

Sender Sent     Receiver Responds   Implication
===============================================
WILL            DO                  The sender would like to use a certain facility if the receiver can handle it. Option is now in effect
WILL            DONT                Receiver says it cannot support the option. Option is not in effect.
DO              WILL                The sender says it can handle traffic from the sender if the sender wishes to use a certain option. Option is now in effect.
DO              WONT                Receiver says it cannot support the option. Option is not in effect.
WONT            DONT                Option disabled. DONT is only valid response.
DONT            WONT                Option disabled. WONT is only valid response.

For example if the sender wants the other end to suppress go-ahead it would send the byte sequence:

    255(IAC),251(WILL),3

The final byte of the three byte sequence identifies the required action.
For some of the negotiable options values need to be communicated once support of the option has
been agreed. This is done using sub-option negotiation. Values are communicated via an exchange of
value query commands and responses in the following form.

    IAC,SB,<option code number>,1,IAC,SE

and

    IAC,SB,<option code>,0,<value>,IAC,SE

For example if the client wishes to identify the terminal type to the server the following exchange
might take place

Client   255(IAC),251(WILL),24
Server   255(IAC),253(DO),24
Server   255(IAC),250(SB),24,1,255(IAC),240(SE)
Client   255(IAC),250(SB),24,0,'V','T','2','2','0',255(IAC),240(SE)

The first exchange establishes that terminal type (option number 24) will be handled, the server
then enquires of the client what value it wishes to associate with the terminal type. The sequence
SB,24,1 implies sub-option negotiation for option type 24, value required (1). The IAC,SE sequence
indicates the end of this request. The repsonse IAC,SB,24,0,'V'... implies sub-option negotiation
for option type 24, value supplied (0), the IAC,SE sequence indicates the end of the response
(and the supplied value). The encoding of the value is specific to the option but a sequence of
characters, as shown above, is common.

Telnet Negotiable Options
=========================
=========================
Many of those listed are self-evident, but some call for more comments.

Suppress Go Ahead
=========================
The original telnet implementation defaulted to "half duplex" operation. This means that data traffic
could only go in one direction at a time and specific action is required to indicate the end of traffic
in one direction and that traffic may now start in the other direction. [This similar to the use of
"roger" and "over" by amateur and CB radio operators.] The specific action is the inclusion of a GA
character in the data stream.

Modern links normally allow bi-directional operation and the "suppress go ahead" option is enabled.

echo
=========================
The echo option is enabled, usually by the server, to indicate that the server will echo every
character it receives. A combination of "suppress go ahead" and "echo" is called character at a time
mode meaning that each character is separately transmitted and echoed.

There is an understanding known as kludge line mode which means that if either "suppress go ahead"
or "echo" is enabled but not both then telnet operates in line at a time mode meaning that complete
lines are assembled at each end and transmitted in one "go".

linemode
=========================
This option replaces and supersedes the line mode kludge.

remote flow control
=========================
This option controls where the special flow control effects of Ctrl-S/Ctrl-Q are implemented.

Telnet control functions
=========================
=========================
The telnet protocol includes a number of control functions. These are initiated in response to
conditions detected by the client (usually certain special keys or key combinations) or server.
The detected condition causes a special character to be incorporated in the data stream.

Interrupt Process
=========================
This is used by the client to cause the suspension or termination of the server process. Typically the
user types Ctrl-C on the keyboard. An IP (244) character is included in the data stream.

Abort Output
=========================
This is used to suppress the transmission of remote process output. An AO (238) character is included
in the data stream.

Are You There
=========================
This is used to trigger a visible response from the other end to confirm the operation of the link and
the remote process. An AYT (246) character is incorporated in the data stream.

Erase character
=========================
Sent to the display to tell it to delete the immediately preceding character from the display. An EC
(247) character is incorporated in the data stream.

Erase line
=========================
Causes the deletion of the current line of input. An EL (248) character is incorporated in the data
stream.

Data Mark
=========================
Some control functions such as AO and IP require immediate action and this may cause difficulties
if data is held in buffers awaiting input requests from a (possibly misbehaving) remote process.
To overcome this problem a DM (242) character is sent in a TCP Urgent segment, this tells the receiver
to examine the data stream for "interesting" characters such as IP, AO and AYT. This is known as the
telnet synch mechanism.

A DM not in a TCP Urgent segment has no effect.
*/
/*EOF*/
```

#### bgXmlRpcParser.c
```c
#ifndef _BG_XMLRPCPARSER_C
#define _BG_XMLRPCPARSER_C

#include "bgXmlRpcParser.h"
#include "bgString.h"

#ifdef WIN32
#include <stdio.h>
#include <string.h>
#define DBGMSG printf
#else
#include "bgSscanf.h"
#endif

/*
##################################################################################
Xml Rpc Parser
##################################################################################
*/
static int	bgXmlRpcFindNextKeyword(char* pSrc, int* isKeywStartOrEnd, char** pBegKeyw, char** pEndKeyw, char* pKeywCopyBuf, int keywCopyBufSize, int* keywLineNo, int* keywColNo);
static int	bgXmlRpcCopyMemBlock(char* pDst, char* pStart, char* pEnd, int destSize, int* copyTrunc);
static int	bgXmlRpcFindKeywordId(char* pKeywStr);

static char* xmlRpcKeywDict[XMLRPC_ID_MAX]={
XMLRPC_STR_ARRAY,
XMLRPC_STR_BASE64,
XMLRPC_STR_BOOL,
XMLRPC_STR_DATA,
XMLRPC_STR_TIME,
XMLRPC_STR_DOUBLE,
XMLRPC_STR_FAULT,
XMLRPC_STR_I4,
XMLRPC_STR_INT,
XMLRPC_STR_METHOD_CALL,
XMLRPC_STR_METHOD_NAME,
XMLRPC_STR_METHOD_RSP,
XMLRPC_STR_MEMBER,
XMLRPC_STR_NAME,
XMLRPC_STR_PARAM,
XMLRPC_STR_PARAMS,
XMLRPC_STR_STRUCT,
XMLRPC_STR_STRING,
XMLRPC_STR_VALUE,
XMLRPC_STR_XMLHEADLINE,
};

char*	bgXmlRpcGetKeywordStr(int keywId)
{
	if(keywId >= XMLRPC_ID_MAX)
		return "not found";

	return xmlRpcKeywDict[keywId];
}

static int bgXmlRpcConvertScalarType(char* valueStr, int keywId)
{
int value;
float fvalue;

	if( (keywId == XMLRPC_ID_I4) ||
		(keywId == XMLRPC_ID_INT)){
		bgsscanf(valueStr, "%d", &value);
		return value;
	}

	if( (keywId == XMLRPC_ID_DOUBLE)){
		bgsscanf(valueStr, "%f", &fvalue);
/*		printf("Float value=%f\n", fvalue);
*/
		return (int)fvalue;
	}

	if( (keywId == XMLRPC_ID_BOOL)){
		char txtBuf[64];
		bgStrCpyNTrimSpcsToLwr(txtBuf, valueStr, 64);
		if( !strcmp(txtBuf, "false") || !strcmp(txtBuf, "0") ){
			value = 0;
		}else{
			value = 1;
		}
		return value;
	}

	return 0;
}

static int	bgXmlRpcFindKeywordId(char* pKeywStr)
{
/*
Return:
>=0 - match id
-1  - match not found
-2  - more then one match
*/
int i;
int j;

int matchList[XMLRPC_ID_MAX];

char* pKeywFromList;
char* pThis = pKeywStr;

int matchId;

    for(i=0;i<XMLRPC_ID_MAX;i++){
        matchList[i] = i;
    }

    j = 0;
    while(1){
        for(i=0;i<XMLRPC_ID_MAX;i++){
            if( matchList[i] >= 0 ){
                pKeywFromList = xmlRpcKeywDict[i];

				if( (*(pThis + j)) == (*(pKeywFromList + j)) )
					matchList[i] = i;
				else
					matchList[i] = -1;
			}
        }

		if( ! (*(pThis + j)) )
			break;

		j++;
    }

    matchId = -1;
    for(i=0;i<XMLRPC_ID_MAX;i++){
        if( matchList[i] >= 0){
            if( matchId < 0)
                matchId = i;
            else
                return -2;
        }
    }

    return matchId;
}

static int	bgXmlRpcCopyMemBlock(char* pDst, char* pStart, char* pEnd, int destSize, int* copyTruncated)
{
int size = pEnd - pStart;

	*copyTruncated = 0;

	if( !pStart || !pEnd || !pDst)
        return 0;

    if( size <= 0 )
        return  0;

	if( size >= destSize ){
        size = destSize;
		*copyTruncated = 1;
	}

    memcpy(pDst, pStart, size);

	pDst[size] = 0;

    return size;
}

static int	bgXmlRpcFindNextKeyword(char* pSrc, int* isKeywStartOrEnd, char** pBegKeyw, char** pEndKeyw, char* pKeywCopyBuf, int keywCopyBufSize,  int* keywLineNo, int* keywColNo)
{
/*search starting position*/
char* p = pSrc;
char* dst = 0;
int len;
static int line = 0;
static int col = 0;

    /*is keyw copy buffer defined?*/
    if(pKeywCopyBuf){
        dst = pKeywCopyBuf;
        *dst = 0;
        len = 0;
    }

	/*initial call*/
	if(!(*pBegKeyw) || !(*pEndKeyw)){
		line = 1;
		col = 1;
	}

    *isKeywStartOrEnd = 0;

    /*find start marker*/
    while(1){
        if( *p == '<' )
            break;

        if( *p == 0 )
            return 1;

		/*increment line & col count*/
		if( *p == '\n'){
			line++;
			col = 1;
		}else{
			col++;
		}

        p++;
    }

    /*found start marker ('<')! it marks the begin of the xml keyword!*/
	*keywLineNo = line;
	*keywColNo = col;

    /*output parametar: start marker ptr*/
    if(pBegKeyw)
        *pBegKeyw = p;

    /*next: advance to the next char*/
    p++;

    /*look for end marker, copy src to dst, look for '/' and don't copy spaces*/
    while(1){
        if( *p == '>' )
            break;

        if( *p == 0 )
            return 1;

        if( *p == '/' ){            /*if end marker, mark a flag*/
            *isKeywStartOrEnd = 1;
        }else
        if( *p == ' ' ){            /*don't copy spaces*/

        }
        else{                       /*copy keyw into supplied buffer*/
            if( dst && (len < (keywCopyBufSize - 1))){
                *dst = *p;
    			dst++;
                len++;
            }
        }

		/*increment line & col count*/
		if( *p == '\n'){
			line++;
			col = 1;
		}else{
			col++;
		}

        p++;
    }

    /*output parametar: end marker ptr*/
    if(pEndKeyw)
        *pEndKeyw = p;

    /*terminate dst buffer that contains a keyword!*/
    if( dst ){
        *dst = 0;

        /*convert copy of the keyw into lowercase*/
        bgStringLower(dst);
    }

#if 0
    /*find what keyword is this*/
    DBGMSG("keyword: %s, %d, pBeg=%p, pEnd=%p\n", pKeywCopyBuf?pKeywCopyBuf:"n/a", *isKeywStartOrEnd, *pBegKeyw, *pEndKeyw);
#endif

	return 0;
}

void bgXmlRpcParserInit(bgXmlRpcParser_typ* p, char *pInputStream, char* pTreeMem, int sizeTreeMem, char* pStringMem, int sizeStringMem)
{
    p->initOk = 0;

    if( !p || !pInputStream || !pTreeMem || !pStringMem)
        return;

    if( (sizeTreeMem < 255) || (sizeStringMem < 255) )
        return;

    p->pInputStream = pInputStream;
    p->pXmlTreeMem = pTreeMem;
    p->sizeXmlTreeMem = sizeTreeMem;
    p->pStrHeapMem = pStringMem;
    p->sizeStrHeapMem = sizeStringMem;

    p->initOk = 1;

}

int bgXmlRpcParserSerialize(bgXmlRpcParser_typ* p)
{

	return 0;
}

static int isItemOnTopOfStack(bgStack_typ* s, int keywId)
{
	if( !bgStackGetItemCount(s) || ( (int)bgStackPeek(s) != keywId) )
		return 0;
	else
		return 1;
}

static void setErrorInfo(bgXmlRpcParser_typ* p, int error, int keywId)
{
	p->error = error;
	p->keywId = keywId;
}

void bgXmlRpcParserParse(bgXmlRpcParser_typ* p)
{
int keywIdStack = 0;
int isBlockEnd = 0;
int isBlockBeg = 0;
char* pSearchStart = p->pInputStream;
char* pKeywStart = 0;
char* pKeywEnd = 0;
char* pBegKeywContent = 0;
bgTree4C_typ* pXmlTree = &p->xmlTree;
bgStack_typ* s = &p->stack;
bgStringHeap_typ* pStrHeap = &p->strHeap;
bgTree4CNode_typ* pXmlNodeCurrent = 0;
bgTree4CNode_typ* pXmlNode = 0;
char keywText[32];

    if(!p->initOk)
        return;

	setErrorInfo(p, 0,0); /*no errors*/
	p->keywLineNo = 0;
	p->keywColNo = 0;
	keywText[0] = 0;

    /*init xml tree*/
	bgTree4CInit(pXmlTree, p->pXmlTreeMem, p->sizeXmlTreeMem);

	/*create root node*/
	if( !(pXmlNodeCurrent = bgTree4CNodeCreate(pXmlTree)) ){
		setErrorInfo(p, XMLRPC_ERROR_NODE_CREATE, 0);
		return;
	}

    /*init stack*/
	bgStackInit(s);

    /*init string heap*/
	bgStringHeapInit(pStrHeap, p->pStrHeapMem, p->sizeStrHeapMem);

    while( !bgXmlRpcFindNextKeyword(pSearchStart, &isBlockEnd, &pKeywStart, &pKeywEnd, keywText, 32, &p->keywLineNo, &p->keywColNo) ){
		char txtBuf[128];
		int cpTrunc;
		int cpLen;
        int keywId;
		char* pStr;

		/*extract/copy keyword text into a private buffer*/
		cpLen = bgXmlRpcCopyMemBlock(txtBuf, (char*)(pKeywStart + 1), pKeywEnd, 128, &cpTrunc);

		/*find keyword id*/
        keywId = bgXmlRpcFindKeywordId(keywText);

		/*begining keyword or ending keyword?*/
		isBlockBeg = isBlockEnd ? 0 : 1;

		/*skip following keywords, not used, not checked*/
        if( (keywId == XMLRPC_ID_PARAMS) ||
			(keywId == XMLRPC_ID_PARAM) ||
			(keywId == XMLRPC_ID_XMLHEADLINE) ){
/*
            DBGMSG("found keyword [%s], isBlockBeg=%d\n", xmlRpcKeywDict[keywId], isBlockBeg);
*/
			pSearchStart = pKeywEnd;
			continue;
        }

/*
		DBGMSG("Current NodeId=%d\n", pXmlNodeCurrent ? pXmlNodeCurrent->id : -1);
*/

		if( bgTree4CGetCountFreeNodes(pXmlTree) <= 2 ){
			setErrorInfo(p, XMLRPC_ERROR_NODE_CREATE, keywId);
			return;
		}

		if(isBlockBeg){

			pBegKeywContent = pKeywEnd + 1;

            switch( keywId ){
                case XMLRPC_ID_METHOD_CALL:
                case XMLRPC_ID_METHOD_NAME:
                case XMLRPC_ID_METHOD_RSP:
                case XMLRPC_ID_VALUE:
					/*create new node*/
					pXmlNode = bgTree4CNodeCreate(pXmlTree);
					/*set node data*/
					bgTree4CNodeSetDataType( pXmlNode, keywId);
					/*connect node to "down" at the bottom end from the current node*/
					bgTree4CNodeAppendToDwEnd(pXmlNodeCurrent, pXmlNode);
					/*set newly created node as the new current node*/
					pXmlNodeCurrent = pXmlNode;
                break;
				case XMLRPC_ID_ARRAY:
                case XMLRPC_ID_STRUCT:
					/*struct, array must be inside the value block*/
					if( !isItemOnTopOfStack(s, XMLRPC_ID_VALUE) ){
						setErrorInfo(p, XMLRPC_ERROR_INVALID_XML_BLOCK1, keywId);
                        return;
					}
					/*create new node*/
					pXmlNode = bgTree4CNodeCreate(pXmlTree);
					/*set node data type*/
					bgTree4CNodeSetDataType(pXmlNode, keywId);
					/*check if the current node has higher level*/
					if(!pXmlNodeCurrent->rt ){
						/*higher level=no; insert new node to the rt, create new level*/
						bgTree4CNodeInsertRt(pXmlNodeCurrent, pXmlNode);
					}else{
						/*higher level=yes; insert new node down, on the same level*/
						bgTree4CNodeAppendToDwEnd(pXmlNodeCurrent, pXmlNode);
					}
					/*set new node as the new current node*/
					pXmlNodeCurrent = pXmlNode;
				break;
                case XMLRPC_ID_MEMBER:
					/*member must be inside struct*/
					if( !isItemOnTopOfStack(s, XMLRPC_ID_STRUCT) ){
						setErrorInfo(p, XMLRPC_ERROR_INVALID_XML_BLOCK2, keywId);
                        return;
					}

					/*create new node*/
					pXmlNode = bgTree4CNodeCreate(pXmlTree);
					/*set node data type*/
					bgTree4CNodeSetDataType(pXmlNode, keywId);
					if(pXmlNodeCurrent->dataType == XMLRPC_ID_STRUCT){
						/*insert new node to the rt, create new level*/
						bgTree4CNodeInsertRt(pXmlNodeCurrent, pXmlNode);
					}else{
						/*insert new node to dw, same level*/
						bgTree4CNodeAppendToDwEnd(pXmlNodeCurrent, pXmlNode);
					}
					/*set new node as the new current node*/
					pXmlNodeCurrent = pXmlNode;
                break;
                case XMLRPC_ID_NAME:
					/*name must be inside member*/
					if( !isItemOnTopOfStack(s, XMLRPC_ID_MEMBER) ){
						setErrorInfo(p, XMLRPC_ERROR_INVALID_XML_BLOCK3, keywId);
                        return;
					}

					/*create new node*/
					pXmlNode = bgTree4CNodeCreate(pXmlTree);
					/*set node data*/
					bgTree4CNodeSetDataType(pXmlNode, keywId);
					/*insert new node to the rt, create new level*/
					bgTree4CNodeInsertRt(pXmlNodeCurrent, pXmlNode);
					/*set new node as the new current node*/
					pXmlNodeCurrent = pXmlNode;
                break;
				case XMLRPC_ID_I4:
				case XMLRPC_ID_DOUBLE:
                case XMLRPC_ID_INT:
                case XMLRPC_ID_STRING:
                case XMLRPC_ID_BOOL:
					/*scalar types must be inside  value*/
					if( !isItemOnTopOfStack(s, XMLRPC_ID_VALUE) ){
						setErrorInfo(p, XMLRPC_ERROR_INVALID_XML_BLOCK4, keywId);
                        return;
					}
					/*create new node*/
					pXmlNode = bgTree4CNodeCreate(pXmlTree);
					/*set node data*/
					bgTree4CNodeSetDataType(pXmlNode, keywId);
					/*highest level nodes > always to the end of the current node*/
					bgTree4CNodeAppendToRtEnd(pXmlNodeCurrent, pXmlNode);
				break;
                default:
                break;
			}

            bgStackPush(s, (char*)(keywId));
/*
            DBGMSG("push= %s\n", xmlRpcKeywDict[keywId]);
*/

		}else{

            keywIdStack = (int)bgStackPop(s);
/*
            DBGMSG("pop= %s\n", xmlRpcKeywDict[keywId]);
*/
/*
			DBGMSG("---------------------------------------------------------------\n");
			bgTree4CPrint(pXmlTree);
			DBGMSG("---------------------------------------------------------------\n");
*/

            if((keywId != XMLRPC_ID_VALUE) && (keywIdStack != keywId)){
				setErrorInfo(p, XMLRPC_ERROR_INVALID_XML_BLOCK6, keywId);
                return;
            }

			switch( keywId ){
                case XMLRPC_ID_METHOD_RSP:
				break;
                case XMLRPC_ID_VALUE:
					/*back to the previous level*/
					pXmlNode = bgTree4CNodePreviousLevel(pXmlNodeCurrent);
					if(pXmlNode)
						pXmlNodeCurrent = pXmlNode;
				break;
				case XMLRPC_ID_ARRAY:
                case XMLRPC_ID_STRUCT:
					/*find next lower level with nodeType = _VALUE*/
					while(1){
						pXmlNode = bgTree4CNodePreviousLevel(pXmlNodeCurrent);

						if(pXmlNode){
							pXmlNodeCurrent = pXmlNode;
						}else{
							setErrorInfo(p, XMLRPC_ERROR_INVALID_XML_BLOCK6, keywId);
	                        return;
						}

						if( pXmlNodeCurrent->dataType == XMLRPC_ID_VALUE )
							break;

					}
				break;
                case XMLRPC_ID_METHOD_NAME:
					/*extract/copy keyword text into a private buffer*/
					cpLen = bgXmlRpcCopyMemBlock(txtBuf, pBegKeywContent, pKeywStart, 128, &cpTrunc);
					pStr = bgStringHeapAddString(pStrHeap, txtBuf);
					bgTree4CNodeSetDataPtr(pXmlNodeCurrent, pStr);
				break;
                case XMLRPC_ID_NAME:
                case XMLRPC_ID_STRING:
                case XMLRPC_ID_TIME:
					/*extract/copy keyword text into a private buffer*/
					cpLen = bgXmlRpcCopyMemBlock(txtBuf, pBegKeywContent, pKeywStart, 128, &cpTrunc);
					/*above types are never "current nodes", they are on the right from the current node (i.e. value)*/
					pXmlNode = pXmlNodeCurrent->rt ? pXmlNodeCurrent->rt : pXmlNodeCurrent;
					pStr = bgStringHeapAddString(pStrHeap, txtBuf);
					bgTree4CNodeSetDataPtr(pXmlNode, pStr);
				break;
                case XMLRPC_ID_I4:
                case XMLRPC_ID_INT:
                case XMLRPC_ID_BOOL:
                case XMLRPC_ID_DOUBLE:
					/*extract/copy keyword text into a private buffer*/
					cpLen = bgXmlRpcCopyMemBlock(txtBuf, pBegKeywContent, pKeywStart, 128, &cpTrunc);
					/*above types are never "current nodes", they are on the right from the current node (i.e. value)*/
					pXmlNode = pXmlNodeCurrent->rt ? pXmlNodeCurrent->rt : pXmlNodeCurrent;
					pStr = bgStringHeapAddString(pStrHeap, txtBuf);
					bgTree4CNodeSetDataPtr(pXmlNode, pStr);

					/*for scalar types, also convert value and store it on the node*/
					bgTree4CNodeSetDataValue(pXmlNode, bgXmlRpcConvertScalarType(txtBuf, keywId));
				break;
                default:
                break;
            }

        }

/*
		DBGMSG("---------------------------------------------------------------\n");
		bgTree4CPrint(pXmlTree);
		DBGMSG("---------------------------------------------------------------\n");
*/
		pSearchStart = pKeywEnd;
    }
	return;
}

#endif
```

### bglibas.typ
```iecst
(********************************************************************
 * COPYRIGHT -- pai
 ********************************************************************
 * Library: bglibas
 * File: bglibas.typ
 * Author: admin
 * Created: March 07, 2012
 ********************************************************************
 * Data types of library bglibas
 ********************************************************************)

TYPE
	BGSSM_CONST_XYZ :
		(
		BGSSM_FLAG_COUNT := 5,
		BGSSM_EVENT_COUNT := 5,
		BGSSM_COUNTER_COUNT := 5,
		BGSSM_TIMER_COUNT := 5,
		BGSSM_REGISTER_COUNT := 5
		);
	bgFIFO_typ : 	STRUCT
		iPtrPushData : UDINT;
		cfgEntrySize : UDINT;
		cfgMaxEntries : UDINT;
		oPtrPullData : UDINT;
		oFIFOCount : UDINT;
		oFIFOFull : UDINT;
		oPushIdx : UDINT;
		oPullIdx : UDINT;
		prvFIFOMemory : UDINT;
	END_STRUCT;
	bgSSM_typ : 	STRUCT
		state : UDINT;
		stateNext : UDINT;
		stateRet : UDINT;
		stateOld : UDINT;
		stateText : STRING[31];
		pfunGetStateName : UDINT;
		pfunCyclicCallback : UDINT;
		stateInit : BOOL;
		error : UDINT;
		errorText : STRING[31];
		event : ARRAY[0..BGSSM_EVENT_COUNT]OF BOOL;
		flag : ARRAY[0..BGSSM_FLAG_COUNT]OF BOOL;
		counter : ARRAY[0..BGSSM_COUNTER_COUNT]OF UDINT;
		value : ARRAY[0..BGSSM_REGISTER_COUNT]OF UDINT;
		timer_x1ms : ARRAY[0..BGSSM_TIMER_COUNT]OF TON;
		dlytimer_x1ms : TON;
		dlyCycles : UDINT;
	END_STRUCT;
END_TYPE
```

- Library Logical/paiComponents/Libraries/bgringbuf (ANSIC) (no source held here)

### paiVFDX64ParRW.var
```iecst
VAR
	gPaiVFDX64Mgr : paiBnRVFDX64RWMgr_typ := (0);
END_VAR
VAR CONSTANT
	paiBnRVFDX64ParamIdxMax : UDINT := 4;
	paiBnRVFDX64DriveIdxMax : UDINT := 10;
END_VAR
```

### Program Logical/paiComponents/paiBnRVFD/paiVFDX64

#### paiVFDX64ParRW.c
```c
#include <bur/plctypes.h>

#ifdef _DEFAULT_INCLUDES
	#include <AsDefault.h>
#endif

static void paiVFDX64ParNextStation()
{
	gPaiVFDX64Mgr.mCurrentEntry++;
	if(gPaiVFDX64Mgr.mCurrentEntry > paiBnRVFDX64DriveIdxMax){
		gPaiVFDX64Mgr.mCurrentEntry = 0;
	}
}

static void paiVFDX64ParNextParam()
{
	int vfdIdx = gPaiVFDX64Mgr.mCurrentEntry;

	gPaiVFDX64Mgr.mX64VFDs[vfdIdx].mCurrentEntry++;
	if(gPaiVFDX64Mgr.mX64VFDs[vfdIdx].mCurrentEntry > paiBnRVFDX64ParamIdxMax){
		gPaiVFDX64Mgr.mX64VFDs[vfdIdx].mCurrentEntry = 0;
		paiVFDX64ParNextStation();
	}
}

static BOOL paiVFDX64IsParamActive(int vfdIdx, int parIdx)
{
BOOL *pModuleOk = 0;

	//check module ok ptr
	if(gPaiVFDX64Mgr.mX64VFDs[vfdIdx].iPtrModuleOk){
		pModuleOk = (BOOL*) gPaiVFDX64Mgr.mX64VFDs[vfdIdx].iPtrModuleOk;
	}

	//device name not defined > skip to next station
	if(!gPaiVFDX64Mgr.mX64VFDs[vfdIdx].iDeviceName[0]){
		gPaiVFDX64Mgr.mX64VFDs[vfdIdx].mX64Params[parIdx].mState = 0;
		paiVFDX64ParNextStation();
		return 0;
	}

	//if module ok ptr defined && module is NOT OK > skip to next vfd station
	if(pModuleOk && !(*pModuleOk)){
		gPaiVFDX64Mgr.mX64VFDs[vfdIdx].mX64Params[parIdx].mState = 0;
		paiVFDX64ParNextStation();
		return 0;
	}

	//if RD channel not defined > skip to next param
	if(	!gPaiVFDX64Mgr.mX64VFDs[vfdIdx].mX64Params[parIdx].iChannelNameRD[0]){
		gPaiVFDX64Mgr.mX64VFDs[vfdIdx].mX64Params[parIdx].mState = 0;
		paiVFDX64ParNextParam();
		return 0;
	}

	return 1;
}

static void paiVFDX64SingleParReadCyclic(int vfdIdx, int parIdx)
{
	gPaiVFDX64Mgr.mAsIOAccRd.enable = 1;
	gPaiVFDX64Mgr.mAsIOAccRd.pDeviceName = (UDINT)&gPaiVFDX64Mgr.mX64VFDs[vfdIdx].iDeviceName;
	gPaiVFDX64Mgr.mAsIOAccRd.pChannelName = (UDINT)&gPaiVFDX64Mgr.mX64VFDs[vfdIdx].mX64Params[parIdx].iChannelNameRD;

	AsIOAccRead( &gPaiVFDX64Mgr.mAsIOAccRd );

	if(gPaiVFDX64Mgr.mAsIOAccRd.status == ERR_FUB_BUSY){
		gPaiVFDX64Mgr.mX64VFDs[vfdIdx].mX64Params[parIdx].mState = 2;
		return;
	}
	gPaiVFDX64Mgr.mX64VFDs[vfdIdx].mX64Params[parIdx].oStatusRD = gPaiVFDX64Mgr.mAsIOAccRd.status;
	gPaiVFDX64Mgr.mX64VFDs[vfdIdx].mX64Params[parIdx].oValue = gPaiVFDX64Mgr.mAsIOAccRd.value;
	if(!gPaiVFDX64Mgr.mAsIOAccRd.status){
		gPaiVFDX64Mgr.mX64VFDs[vfdIdx].mX64Params[parIdx].mState = 1; //upon sucessful RD, go to idle
	}else{
		gPaiVFDX64Mgr.mX64VFDs[vfdIdx].mX64Params[parIdx].mState = 2;//try read again
		paiVFDX64ParNextParam();
	}
}

static void paiVFDX64SingleParWriteCyclic(int vfdIdx, int parIdx)
{
	gPaiVFDX64Mgr.mAsIOAccWr.enable = 1;
	gPaiVFDX64Mgr.mAsIOAccWr.pDeviceName = (UDINT)&gPaiVFDX64Mgr.mX64VFDs[vfdIdx].iDeviceName;
	gPaiVFDX64Mgr.mAsIOAccWr.pChannelName = (UDINT)&gPaiVFDX64Mgr.mX64VFDs[vfdIdx].mX64Params[parIdx].iChannelNameWR;
	gPaiVFDX64Mgr.mAsIOAccWr.value = (UDINT)gPaiVFDX64Mgr.mX64VFDs[vfdIdx].mX64Params[parIdx].iValueWR;

	AsIOAccWrite( &gPaiVFDX64Mgr.mAsIOAccWr );

	if(gPaiVFDX64Mgr.mAsIOAccWr.status == ERR_FUB_BUSY){
		gPaiVFDX64Mgr.mX64VFDs[vfdIdx].mX64Params[parIdx].mState = 3;
		return;
	}
	gPaiVFDX64Mgr.mX64VFDs[vfdIdx].mX64Params[parIdx].oStatusWR = gPaiVFDX64Mgr.mAsIOAccWr.status;
	if(!gPaiVFDX64Mgr.mAsIOAccWr.status){
		gPaiVFDX64Mgr.mX64VFDs[vfdIdx].mX64Params[parIdx].mState = 2;//upon successful WR trigger RD
		paiVFDX64ParNextParam();
	}else{
		gPaiVFDX64Mgr.mX64VFDs[vfdIdx].mX64Params[parIdx].mState = 1;
	}
}

static void paiVFDX64ParamRWCyclic()
{
	int vfdIdx = gPaiVFDX64Mgr.mCurrentEntry;
	int parIdx = gPaiVFDX64Mgr.mX64VFDs[vfdIdx].mCurrentEntry;

	if( !paiVFDX64IsParamActive(vfdIdx, parIdx) ){
		return;
	}

	//Param access state machine
	//0-init not completed, RD needed
	//1-idle
	//2-rd in progress
	//3-wr in progress
	switch(gPaiVFDX64Mgr.mX64VFDs[vfdIdx].mX64Params[parIdx].mState){
		case 0:
			//init
			gPaiVFDX64Mgr.mX64VFDs[vfdIdx].mX64Params[parIdx].mState = 2;//activate RD
			break;
		case 1:
			//idle(rd not required)
			gPaiVFDX64Mgr.mAsIOAccRd.enable = 0;
			AsIOAccRead( &gPaiVFDX64Mgr.mAsIOAccRd );

			gPaiVFDX64Mgr.mAsIOAccWr.enable = 0;
			AsIOAccWrite( &gPaiVFDX64Mgr.mAsIOAccWr );

			//check if write required?
			if(gPaiVFDX64Mgr.mX64VFDs[vfdIdx].mX64Params[parIdx].oValue != gPaiVFDX64Mgr.mX64VFDs[vfdIdx].mX64Params[parIdx].iValueWR){
				//write is required
				gPaiVFDX64Mgr.mX64VFDs[vfdIdx].mX64Params[parIdx].mState = 3;//activate WR
			}
			//process next item
			paiVFDX64ParNextParam();
			return;
			break;
		case 2:
			//read in progress
			paiVFDX64SingleParReadCyclic(vfdIdx, parIdx);
			break;
		case 3:
			//write in progress
			paiVFDX64SingleParWriteCyclic(vfdIdx, parIdx);
			break;
		default:
			return;
			break;
	}
}

static void paiVFDX64ParamConfigWrite()
{
	//Copy configuration parameters from the config to the VFD WR parameter channel

#if 0
	//VFD accelration
	gPaiVFDX64Mgr.mX64VFDs[0].mX64Params[0].iValueWR = gConfigApp.vfd[1].acc;
	gPaiVFDX64Mgr.mX64VFDs[1].mX64Params[0].iValueWR = gConfigApp.vfd[2].acc;
	gPaiVFDX64Mgr.mX64VFDs[2].mX64Params[0].iValueWR = gConfigApp.vfd[5].acc;
	gPaiVFDX64Mgr.mX64VFDs[3].mX64Params[0].iValueWR = gConfigApp.vfd[6].acc;
	gPaiVFDX64Mgr.mX64VFDs[4].mX64Params[0].iValueWR = gConfigApp.vfd[11].acc;
	gPaiVFDX64Mgr.mX64VFDs[5].mX64Params[0].iValueWR = gConfigApp.vfd[12].acc;

	//VFD deceleration
	gPaiVFDX64Mgr.mX64VFDs[0].mX64Params[1].iValueWR = gConfigApp.vfd[1].dec;
	gPaiVFDX64Mgr.mX64VFDs[1].mX64Params[1].iValueWR = gConfigApp.vfd[2].dec;
	gPaiVFDX64Mgr.mX64VFDs[2].mX64Params[1].iValueWR = gConfigApp.vfd[5].dec;
	gPaiVFDX64Mgr.mX64VFDs[3].mX64Params[1].iValueWR = gConfigApp.vfd[6].dec;
	gPaiVFDX64Mgr.mX64VFDs[4].mX64Params[1].iValueWR = gConfigApp.vfd[11].dec;
	gPaiVFDX64Mgr.mX64VFDs[5].mX64Params[1].iValueWR = gConfigApp.vfd[12].dec;
#endif

	//VFD accelration
	gPaiVFDX64Mgr.mX64VFDs[0].mX64Params[0].iValueWR = gPallete.palCfg.palSettings.vfd[1].acc;
	gPaiVFDX64Mgr.mX64VFDs[1].mX64Params[0].iValueWR = gPallete.palCfg.palSettings.vfd[2].acc;
	gPaiVFDX64Mgr.mX64VFDs[2].mX64Params[0].iValueWR = gPallete.palCfg.palSettings.vfd[5].acc;
	gPaiVFDX64Mgr.mX64VFDs[3].mX64Params[0].iValueWR = gPallete.palCfg.palSettings.vfd[6].acc;
	gPaiVFDX64Mgr.mX64VFDs[4].mX64Params[0].iValueWR = gPallete.palCfg.palSettings.vfd[11].acc;
	gPaiVFDX64Mgr.mX64VFDs[5].mX64Params[0].iValueWR = gPallete.palCfg.palSettings.vfd[12].acc;

	//VFD deceleration
	gPaiVFDX64Mgr.mX64VFDs[0].mX64Params[1].iValueWR = gPallete.palCfg.palSettings.vfd[1].dec;
	gPaiVFDX64Mgr.mX64VFDs[1].mX64Params[1].iValueWR = gPallete.palCfg.palSettings.vfd[2].dec;
	gPaiVFDX64Mgr.mX64VFDs[2].mX64Params[1].iValueWR = gPallete.palCfg.palSettings.vfd[5].dec;
	gPaiVFDX64Mgr.mX64VFDs[3].mX64Params[1].iValueWR = gPallete.palCfg.palSettings.vfd[6].dec;
	gPaiVFDX64Mgr.mX64VFDs[4].mX64Params[1].iValueWR = gPallete.palCfg.palSettings.vfd[11].dec;
	gPaiVFDX64Mgr.mX64VFDs[5].mX64Params[1].iValueWR = gPallete.palCfg.palSettings.vfd[12].dec;

}

void _INIT paiVFDX64ParRWInit(void)
{
	// Insert code here

	brsstrcpy((UDINT)&gPaiVFDX64Mgr.mX64VFDs[0].iDeviceName, (UDINT)"IF5.ST9");
	brsstrcpy((UDINT)&gPaiVFDX64Mgr.mX64VFDs[0].iDescription, (UDINT)"VFD1");
	gPaiVFDX64Mgr.mX64VFDs[0].iPtrModuleOk = (UDINT)&gHWModules[9].ModuleOk;
	brsstrcpy((UDINT)&gPaiVFDX64Mgr.mX64VFDs[0].mX64Params[0].iChannelNameRD , (UDINT)"ACC_Input");
	brsstrcpy((UDINT)&gPaiVFDX64Mgr.mX64VFDs[0].mX64Params[0].iChannelNameWR , (UDINT)"ACC_Output");
	brsstrcpy((UDINT)&gPaiVFDX64Mgr.mX64VFDs[0].mX64Params[1].iChannelNameRD , (UDINT)"DEC_Input");
	brsstrcpy((UDINT)&gPaiVFDX64Mgr.mX64VFDs[0].mX64Params[1].iChannelNameWR , (UDINT)"DEC_Output");

	brsstrcpy((UDINT)&gPaiVFDX64Mgr.mX64VFDs[1].iDeviceName, (UDINT)"IF5.ST10");
	brsstrcpy((UDINT)&gPaiVFDX64Mgr.mX64VFDs[1].iDescription, (UDINT)"VFD2");
	gPaiVFDX64Mgr.mX64VFDs[1].iPtrModuleOk = (UDINT)&gHWModules[10].ModuleOk;
	brsstrcpy((UDINT)&gPaiVFDX64Mgr.mX64VFDs[1].mX64Params[0].iChannelNameRD , (UDINT)"ACC_Input");
	brsstrcpy((UDINT)&gPaiVFDX64Mgr.mX64VFDs[1].mX64Params[0].iChannelNameWR , (UDINT)"ACC_Output");
	brsstrcpy((UDINT)&gPaiVFDX64Mgr.mX64VFDs[1].mX64Params[1].iChannelNameRD , (UDINT)"DEC_Input");
	brsstrcpy((UDINT)&gPaiVFDX64Mgr.mX64VFDs[1].mX64Params[1].iChannelNameWR , (UDINT)"DEC_Output");

	brsstrcpy((UDINT)&gPaiVFDX64Mgr.mX64VFDs[2].iDeviceName, (UDINT)"IF5.ST11");
	brsstrcpy((UDINT)&gPaiVFDX64Mgr.mX64VFDs[2].iDescription, (UDINT)"VFD5");
	gPaiVFDX64Mgr.mX64VFDs[2].iPtrModuleOk = (UDINT)&gHWModules[11].ModuleOk;
	brsstrcpy((UDINT)&gPaiVFDX64Mgr.mX64VFDs[2].mX64Params[0].iChannelNameRD , (UDINT)"ACC_Input");
	brsstrcpy((UDINT)&gPaiVFDX64Mgr.mX64VFDs[2].mX64Params[0].iChannelNameWR , (UDINT)"ACC_Output");
	brsstrcpy((UDINT)&gPaiVFDX64Mgr.mX64VFDs[2].mX64Params[1].iChannelNameRD , (UDINT)"DEC_Input");
	brsstrcpy((UDINT)&gPaiVFDX64Mgr.mX64VFDs[2].mX64Params[1].iChannelNameWR , (UDINT)"DEC_Output");

	brsstrcpy((UDINT)&gPaiVFDX64Mgr.mX64VFDs[3].iDeviceName, (UDINT)"IF5.ST12");
	brsstrcpy((UDINT)&gPaiVFDX64Mgr.mX64VFDs[3].iDescription, (UDINT)"VFD52");
	gPaiVFDX64Mgr.mX64VFDs[3].iPtrModuleOk = (UDINT)&gHWModules[12].ModuleOk;
	brsstrcpy((UDINT)&gPaiVFDX64Mgr.mX64VFDs[3].mX64Params[0].iChannelNameRD , (UDINT)"ACC_Input");
	brsstrcpy((UDINT)&gPaiVFDX64Mgr.mX64VFDs[3].mX64Params[0].iChannelNameWR , (UDINT)"ACC_Output");
	brsstrcpy((UDINT)&gPaiVFDX64Mgr.mX64VFDs[3].mX64Params[1].iChannelNameRD , (UDINT)"DEC_Input");
	brsstrcpy((UDINT)&gPaiVFDX64Mgr.mX64VFDs[3].mX64Params[1].iChannelNameWR , (UDINT)"DEC_Output");

	brsstrcpy((UDINT)&gPaiVFDX64Mgr.mX64VFDs[4].iDeviceName, (UDINT)"IF5.ST13");
	brsstrcpy((UDINT)&gPaiVFDX64Mgr.mX64VFDs[4].iDescription, (UDINT)"VFD11");
	gPaiVFDX64Mgr.mX64VFDs[4].iPtrModuleOk = (UDINT)&gHWModules[13].ModuleOk;
	brsstrcpy((UDINT)&gPaiVFDX64Mgr.mX64VFDs[4].mX64Params[0].iChannelNameRD , (UDINT)"ACC_Input");
	brsstrcpy((UDINT)&gPaiVFDX64Mgr.mX64VFDs[4].mX64Params[0].iChannelNameWR , (UDINT)"ACC_Output");
	brsstrcpy((UDINT)&gPaiVFDX64Mgr.mX64VFDs[4].mX64Params[1].iChannelNameRD , (UDINT)"DEC_Input");
	brsstrcpy((UDINT)&gPaiVFDX64Mgr.mX64VFDs[4].mX64Params[1].iChannelNameWR , (UDINT)"DEC_Output");

	brsstrcpy((UDINT)&gPaiVFDX64Mgr.mX64VFDs[5].iDeviceName, (UDINT)"IF5.ST14");
	brsstrcpy((UDINT)&gPaiVFDX64Mgr.mX64VFDs[5].iDescription, (UDINT)"VFD12");
	gPaiVFDX64Mgr.mX64VFDs[5].iPtrModuleOk = (UDINT)&gHWModules[14].ModuleOk;
	brsstrcpy((UDINT)&gPaiVFDX64Mgr.mX64VFDs[5].mX64Params[0].iChannelNameRD , (UDINT)"ACC_Input");
	brsstrcpy((UDINT)&gPaiVFDX64Mgr.mX64VFDs[5].mX64Params[0].iChannelNameWR , (UDINT)"ACC_Output");
	brsstrcpy((UDINT)&gPaiVFDX64Mgr.mX64VFDs[5].mX64Params[1].iChannelNameRD , (UDINT)"DEC_Input");
	brsstrcpy((UDINT)&gPaiVFDX64Mgr.mX64VFDs[5].mX64Params[1].iChannelNameWR , (UDINT)"DEC_Output");
}

void _CYCLIC paiVFDX64ParRWCyclic(void)
{
	// Insert code here

	paiVFDX64ParamConfigWrite();

	paiVFDX64ParamRWCyclic();
}
//eof
```

### paiHmiDialog.typ
```iecst
(********************************************************************
 * COPYRIGHT -- pai
 ********************************************************************
 * Package: HMI
 * File: HMI.typ
 * Author: goran
 * Created: August 28, 2013
 ********************************************************************
 * Data types of package HMI
 ********************************************************************)
(*########################################################################*)
(*HMI object - DIALOG (OK, Cancel)*)
(*########################################################################*)

TYPE
	paiHmiDialog_typ : 	STRUCT
		message : STRING[512];
		result : UINT; (*value returned when button pressed (0-busy, button not pressed, dialog active, OK pressed returns resultForOk (eg.1); Cancel pressed returns resultForCancel (eg.2)*)
		resultForOk : UINT; (*value to return when Ok pressed (if 0 return value is 1)*)
		resultForCancel : UINT; (*value to return when Cancel pressed (if 0 return value is 2)*)
		timeoutConfig : UINT; (*configuration input that defines meaning of the timeout. If 0 > timeout means cancel; if 1> timeout means ok*)
		status : UINT; (*Status for common dialog layer*)
		tmr1RemainingTimeSec : UDINT; (*Timer remaining time (sec)*)
		tmr1 : TON; (*Dialog control timer*)
	END_STRUCT;
END_TYPE
```

### paiHmiDropdownMenuRT.h
```c
/********************************************************************
 * COPYRIGHT --
 ********************************************************************
 * Package: paiHmiTemplate
 * File: paiHmiDropdownMenuRT.h
 * Author: goran
 * Created: July 29, 2015
 *******************************************************************/

#include <bur/plctypes.h>
#ifdef _DEFAULT_INCLUDES
	#include <AsDefault.h>
#endif

//logic control of the global MENU KEYS on the Left Side (i.e. STOPPED, FILLING, PRODUCTION, ...)
void paiHmiDropDownMenuRTInit(paiHmiDropdwMenuRT_typ* p);
//logic control of the global MENU KEYS on the Left Side (i.e. STOPPED, FILLING, PRODUCTION, ...)
void paiHmiDropDownMenuRTCyclic(paiHmiDropdwMenuRT_typ *p);
```

### paiHmiLFMenuTabsPages.h
```c
/********************************************************************
 * COPYRIGHT --
 ********************************************************************
 * Package: paiHmiTemplate
 * File: paiHmiTemplateLogic.c
 * Author: goran
 * Created: July 27, 2015
 *******************************************************************/

#include <bur/plctypes.h>
#ifdef _DEFAULT_INCLUDES
	#include <AsDefault.h>
#endif

void paiHmiPageNavLFMenuTabsCyclic(paiHmiTemplate_typ* p, char* pVisuName, UDINT indexOfTGForHmiNavigation);
```

### paiPingService.typ
```iecst
(********************************************************************
 * COPYRIGHT --
 ********************************************************************
 * Program: paiPingService
 * File: paiPingService.typ
 * Author: goran
 * Created: August 17, 2015
 ********************************************************************
 * Local data types of program paiPingService
 ********************************************************************)

TYPE
	paiPing_typ : 	STRUCT
		iEnable : BOOL;
		iNewIpAddr : BOOL;
		iIPAddrStr : STRING[31];
		iNumericIpAddr : ARRAY[0..3]OF USINT;
		iPingIntervalxms : UDINT;
		iPingTimeoutxms : UDINT;
		oPingOk : BOOL;
		oPingStatus : UDINT; (*0-ping off;1-ping NOT ok; 2-ping ok > connect to a text group to display status*)
		mState : UDINT;
		mPingTimer : TON;
		mIcmpPing : IcmpPing;
	END_STRUCT;
END_TYPE
```

### paiTelnet.typ
```iecst
(********************************************************************
 * COPYRIGHT --
 ********************************************************************
 * Package: paiTelnet
 * File: paiTelnet.typ
 * Author: goran
 * Created: June 23, 2015
 ********************************************************************
 * Data types of package paiTelnet
 ********************************************************************)

TYPE
	bgSocketServerCounter_typ : 	STRUCT
		recv_frames : UDINT;
		iac : UDINT;
		lines : UDINT;
		send_frames : UDINT;
	END_STRUCT;
	bgSocketServer_typ : 	STRUCT
		sockStateData : UINT;
		telnetRecvState : UINT;
		telnetSendState : UINT;
		sockSendOk : UINT;
		cmdError : INT;
		isConnected : BOOL;
		isLoggedIn : BOOL;
		isDataPortReady : BOOL;
		isEcho : BOOL;
		sockData_Timer : UINT;
		sockData_TimerTime : INT;
		sockData_TimerCounter : INT;
		dataRecvBuf : REFERENCE TO SINT;
		dataSendBuf : REFERENCE TO SINT;
		lineRecvBuf : REFERENCE TO SINT;
		ringDataBuffer : UDINT;
		sendRecvBuffer : UDINT;
		iacRecvBuf : ARRAY[0..9]OF SINT;
		New_Member3 : USINT;
		lineIndex : DINT;
		lineIndexPrev : DINT;
		TCPopen_1 : TcpOpen;
		TCPserv_1 : TcpServer;
		TCPsend_1 : TcpSend;
		TCPrecv_1 : TcpRecv;
		TCPclose_1 : TcpClose;
		TCPioctl_1 : TcpIoctl;
		MEMInfo : MEMInfo;
		memAllocStatus1 : UINT;
		memAllocStatus2 : UINT;
		counter : bgSocketServerCounter_typ;
		clientIpAddr : STRING[32];
		delayCounter : INT;
		test : INT;
		testCounter : INT;
		pRB : UDINT;
		New_Member : USINT;
	END_STRUCT;
END_TYPE
```

### paiTelnet.var
```iecst
(********************************************************************
 * COPYRIGHT --
 ********************************************************************
 * Package: paiTelnet
 * File: paiTelnet.var
 * Author: goran
 * Created: June 23, 2015
 ********************************************************************
 * Variables of package paiTelnet
 ********************************************************************)
VAR
	dbgTerm : bgSocketServer_typ := (0);
END_VAR
```

- Visualisation Logical/paiComponents/paiTemplate/paiHMI/paiScreens/paXGA (not shown)

### Program Logical/ParameterDownload/CSV_File

#### SearchFileName.ab
```automation-basic
FUNCTION_BLOCK SearchFileName
;*****************************************************************
;FUB: 			CSV_SearchFileName
;*****************************************************************
;Discription:
;	This FUB search the specified device for the specified file.
;
;Parameter:
;
;Author:	Georg Kreil
;			B&R Eggelsberg
;
;History:	V0.01.6 - 21 July 2003
;					created
;			V0.01.7 - 7 August 2003
;					no changes
;			V0.01.8 - 8 August 2003
;					no changes
;			V0.01.9 - 11 August 2003
;					no changes
;
;*****************************************************************
 select step

;############################################################################################
 	state WAIT
;############################################################################################
 		when(pFileName <> 0) do
 			strcpy(adr(FileName),pFileName)

			loop i=0 to usint(strlen(adr(FileName))) do
				SearchChar access adr(FileName)+i
				exitif(SearchChar = '.')
			endloop

			if(SearchChar <> '.') then
				strcat(adr(FileName), ".CSV")
			endif
			status= 65535
 		next FILEOPEN

;############################################################################################
 	state FILEOPEN
;############################################################################################
		FileOpen_01.enable= 1
		FileOpen_01.pDevice= pDevice
		FileOpen_01.pFile= adr(FileName)
		FileOpen_01.mode= 0
		FileOpen_01 FUB FileOpen()

		when (FileOpen_01.status = 0) do
			status= 65535
		next FILECLOSE

		when (FileOpen_01.status = 65535) do
			status= FileOpen_01.status
		next FILEOPEN

		when (FileOpen_01.status = 20708) do
			status= FILE_NOT_FOUND
		next WAIT

		when (FileOpen_01.status <> 20708) and (FileOpen_01.status <> 0)and (FileOpen_01.status <> 65535) do
			status= FileOpen_01.status
		next WAIT

;############################################################################################
 	state FILECLOSE
;############################################################################################
		FileClose_01.enable= 1
		FileClose_01.ident= FileOpen_01.ident
		FileClose_01 FUB FileClose()

		when (FileClose_01.status = 0) do
			status= FILE_FOUND
		next WAIT

		when (FileClose_01.status = 65535) do
			status= FileClose_01.status
		next FILECLOSE

		when (FileClose_01.status <> 0)and (FileClose_01.status <> 65535) do
			status= FileClose_01.status
		next WAIT

endselect
END_FUNCTION_BLOCK
```

- Program Logical/ParameterDownload/X64_S44_Download/X64param (IEC) (no source held here)

Listed in the project but not available here: Logical/MachineControl/palletinfdis/Cyclic.ld, Logical/MachineControl/palletinfdis/Init.ld, Logical/paiComponents/Libraries/bgringbuf/bgringbuffer.h, Logical/paiComponents/Libraries/bgringbuf/bgringbuffer.c, Logical/ParameterDownload/X64_S44_Download/X64param/X64paramCyclic.st, Logical/ParameterDownload/X64_S44_Download/X64param/X64paramInit.st, Logical/ParameterDownload/X64_S44_Download/X64param/X64param.typ, Logical/ParameterDownload/X64_S44_Download/X64param/X64param.var
